  MoveL 654 to (53.54, -49.32, -190) mm, rotated rx 43.39 ry 15.84 rz 65.61 deg; joints [-1.413, -9.575, 78.286, 154.561, 95.246, 24.079, 178.286]
  MoveL 655 to (54.01, -49.44, -189.99) mm, rotated rx 43.39 ry 15.84 rz 65.61 deg; joints [-1.428, -9.587, 78.293, 154.547, 95.245, 24.086, 178.286]
  MoveL 656 to (54.51, -49.57, -189.99) mm, rotated rx 43.39 ry 15.84 rz 65.61 deg; joints [-1.445, -9.599, 78.299, 154.532, 95.243, 24.093, 178.286]
  MoveL 657 to (55.01, -49.69, -189.98) mm, rotated rx 43.39 ry 15.84 rz 65.61 deg; joints [-1.461, -9.611, 78.308, 154.518, 95.241, 24.101, 178.286]
  MoveL 658 to (55.49, -49.8, -189.95) mm, rotated rx 43.39 ry 15.84 rz 65.61 deg; joints [-1.477, -9.625, 78.317, 154.504, 95.24, 24.107, 178.286]
  MoveL 659 to (55.99, -49.92, -189.94) mm, rotated rx 43.39 ry 15.84 rz 65.61 deg; joints [-1.494, -9.637, 78.325, 154.489, 95.239, 24.115, 178.286]
  MoveL 660 to (58.53, -50.59, -189.94) mm, rotated rx 43.39 ry 15.84 rz 65.61 deg; joints [-1.578, -9.696, 78.356, 154.414, 95.227, 24.155, 178.286]
  MoveL 661 to (59.92, -51.02, -190.02) mm, rotated rx 43.39 ry 15.84 rz 65.61 deg; joints [-1.625, -9.722, 78.36, 154.372, 95.215, 24.18, 178.286]
  MoveL 662 to (61.01, -51.51, -190.27) mm, rotated rx 43.39 ry 15.84 rz 65.61 deg; joints [-1.665, -9.727, 78.336, 154.337, 95.194, 24.206, 178.286]
  MoveL 663 to (61.81, -52.06, -190.69) mm, rotated rx 43.39 ry 15.84 rz 65.61 deg; joints [-1.698, -9.714, 78.284, 154.31, 95.165, 24.233, 178.286]
  MoveL 664 to (62.32, -52.66, -191.27) mm, rotated rx 43.39 ry 15.84 rz 65.61 deg; joints [-1.723, -9.68, 78.204, 154.289, 95.127, 24.262, 178.286]
  MoveL 665 to (62.53, -53.32, -192.02) mm, rotated rx 43.39 ry 15.84 rz 65.61 deg; joints [-1.74, -9.627, 78.096, 154.275, 95.08, 24.292, 178.286]
  MoveL 666 to (62.45, -54.04, -192.93) mm, rotated rx 43.39 ry 15.84 rz 65.61 deg; joints [-1.751, -9.554, 77.959, 154.268, 95.024, 24.323, 178.286]
  MoveL 667 to (61.4, -55.64, -195.26) mm, rotated rx 43.39 ry 15.84 rz 65.61 deg; joints [-1.749, -9.349, 77.601, 154.276, 94.886, 24.389, 178.286]
  MoveL 668 to (59.59, -57.02, -197.61) mm, rotated rx 43.39 ry 15.84 rz 65.61 deg; joints [-1.722, -9.124, 77.232, 154.305, 94.752, 24.443, 178.286]
  MoveL 669 to (57.44, -57.73, -199.32) mm, rotated rx 43.39 ry 15.84 rz 65.61 deg; joints [-1.675, -8.942, 76.96, 154.351, 94.662, 24.466, 178.286]
  MoveL 670 to (56.23, -57.83, -199.93) mm, rotated rx 43.39 ry 15.84 rz 65.61 deg; joints [-1.643, -8.868, 76.859, 154.38, 94.635, 24.466, 178.286]
  MoveL 671 to (54.93, -57.77, -200.39) mm, rotated rx 43.39 ry 15.84 rz 65.61 deg; joints [-1.607, -8.803, 76.783, 154.413, 94.618, 24.459, 178.286]
  MoveL 672 to (52.09, -57.13, -200.82) mm, rotated rx 43.39 ry 15.84 rz 65.61 deg; joints [-1.518, -8.707, 76.704, 154.492, 94.619, 24.422, 178.286]
  MoveL 673 to (51.13, -56.82, -200.85) mm, rotated rx 43.39 ry 15.84 rz 65.61 deg; joints [-1.487, -8.683, 76.694, 154.52, 94.627, 24.405, 178.286]
  MoveL 674 to (48.7, -55.83, -200.85) mm, rotated rx 43.39 ry 15.84 rz 65.61 deg; joints [-1.406, -8.632, 76.694, 154.591, 94.659, 24.356, 178.286]
  MoveL 675 to (47.75, -55.49, -200.91) mm, rotated rx 43.39 ry 15.84 rz 65.61 deg; joints [-1.376, -8.608, 76.685, 154.618, 94.669, 24.339, 178.286]
  MoveL 676 to (46.78, -55.1, -200.91) mm, rotated rx 43.39 ry 15.84 rz 65.61 deg; joints [-1.343, -8.587, 76.685, 154.646, 94.682, 24.319, 178.286]
  MoveL 677 to (46.33, -54.92, -200.92) mm, rotated rx 43.39 ry 15.84 rz 65.61 deg; joints [-1.328, -8.577, 76.683, 154.66, 94.687, 24.31, 178.286]
  MoveL 678 to (45.93, -54.78, -200.94) mm, rotated rx 43.39 ry 15.84 rz 65.61 deg; joints [-1.315, -8.566, 76.679, 154.671, 94.691, 24.303, 178.286]
  MoveL 679 to (45.49, -54.62, -200.95) mm, rotated rx 43.39 ry 15.84 rz 65.61 deg; joints [-1.301, -8.556, 76.677, 154.684, 94.696, 24.295, 178.286]
  MoveL 680 to (43.06, -53.64, -200.96) mm, rotated rx 43.39 ry 15.84 rz 65.61 deg; joints [-1.22, -8.504, 76.675, 154.755, 94.728, 24.246, 178.286]
  MoveL 681 to (42.6, -53.46, -200.98) mm, rotated rx 43.39 ry 15.84 rz 65.61 deg; joints [-1.205, -8.493, 76.672, 154.768, 94.733, 24.238, 178.286]
  MoveL 682 to (42.16, -53.33, -201.02) mm, rotated rx 43.39 ry 15.84 rz 65.61 deg; joints [-1.191, -8.48, 76.664, 154.781, 94.736, 24.231, 178.286]
  MoveL 683 to (41.73, -53.23, -201.06) mm, rotated rx 43.39 ry 15.84 rz 65.61 deg; joints [-1.177, -8.467, 76.654, 154.793, 94.736, 24.225, 178.286]
  MoveL 684 to (41.3, -53.17, -201.09) mm, rotated rx 43.39 ry 15.84 rz 65.61 deg; joints [-1.163, -8.454, 76.641, 154.805, 94.734, 24.22, 178.286]
  MoveL 685 to (40.86, -53.17, -201.11) mm, rotated rx 43.39 ry 15.84 rz 65.61 deg; joints [-1.149, -8.441, 76.624, 154.818, 94.728, 24.217, 178.286]
  MoveL 686 to (40.42, -53.22, -201.11) mm, rotated rx 43.39 ry 15.84 rz 65.61 deg; joints [-1.135, -8.428, 76.603, 154.831, 94.719, 24.216, 178.286]
  MoveL 687 to (41.18, -53.27, -201.85) mm, rotated rx 43.39 ry 15.84 rz 65.61 deg; joints [-1.169, -8.398, 76.567, 154.8, 94.718, 24.23, 178.286]
  MoveL 688 to (39.84, -53.8, -202.4) mm, rotated rx 43.39 ry 15.84 rz 65.61 deg; joints [-1.134, -8.317, 76.427, 154.834, 94.66, 24.243, 178.286]
  MoveL 689 to (38.37, -54.3, -202.83) mm, rotated rx 43.39 ry 15.84 rz 65.61 deg; joints [-1.092, -8.241, 76.296, 154.874, 94.603, 24.253, 178.286]
  MoveL 690 to (36.66, -54.77, -203.13) mm, rotated rx 43.39 ry 15.84 rz 65.61 deg; joints [-1.042, -8.167, 76.166, 154.921, 94.545, 24.259, 178.286]
  MoveL 691 to (34.69, -55.23, -203.32) mm, rotated rx 43.39 ry 15.84 rz 65.61 deg; joints [-0.981, -8.093, 76.038, 154.978, 94.486, 24.261, 178.286]
  MoveL 692 to (32.65, -55.69, -203.51) mm, rotated rx 43.39 ry 15.84 rz 65.61 deg; joints [-0.918, -8.017, 75.905, 155.036, 94.424, 24.264, 178.286]
  MoveL 693 to (30.56, -56.15, -203.63) mm, rotated rx 43.39 ry 15.84 rz 65.61 deg; joints [-0.853, -7.945, 75.777, 155.097, 94.364, 24.265, 178.286]
  MoveL 694 to (28.48, -56.61, -203.86) mm, rotated rx 43.39 ry 15.84 rz 65.61 deg; joints [-0.789, -7.864, 75.639, 155.156, 94.301, 24.268, 178.286]
  MoveL 695 to (26.39, -57.06, -203.97) mm, rotated rx 43.39 ry 15.84 rz 65.61 deg; joints [-0.724, -7.792, 75.511, 155.216, 94.24, 24.268, 178.286]
  MoveL 696 to (24.31, -57.5, -204.09) mm, rotated rx 43.39 ry 15.84 rz 65.61 deg; joints [-0.659, -7.719, 75.382, 155.277, 94.179, 24.269, 178.286]
  MoveL 697 to (22.22, -57.95, -204.21) mm, rotated rx 43.39 ry 15.84 rz 65.61 deg; joints [-0.593, -7.646, 75.254, 155.337, 94.118, 24.27, 178.286]
  MoveL 698 to (20.13, -58.39, -204.44) mm, rotated rx 43.39 ry 15.84 rz 65.61 deg; joints [-0.53, -7.565, 75.115, 155.396, 94.056, 24.272, 178.286]
  MoveL 699 to (18.04, -58.83, -204.56) mm, rotated rx 43.39 ry 15.84 rz 65.61 deg; joints [-0.465, -7.491, 74.985, 155.456, 93.994, 24.273, 178.286]
  MoveL 700 to (16.05, -59.31, -204.67) mm, rotated rx 43.39 ry 15.84 rz 65.61 deg; joints [-0.403, -7.421, 74.856, 155.514, 93.931, 24.275, 178.286]
  MoveL 701 to (14.12, -59.88, -204.87) mm, rotated rx 43.39 ry 15.84 rz 65.61 deg; joints [-0.345, -7.343, 74.712, 155.568, 93.862, 24.283, 178.286]
  MoveL 702 to (11.66, -60.37, -205.01) mm, rotated rx 43.39 ry 15.84 rz 65.61 deg; joints [-0.268, -7.257, 74.561, 155.638, 93.79, 24.282, 178.286]
  MoveL 703 to (9.24, -60.72, -205.09) mm, rotated rx 43.39 ry 15.84 rz 65.61 deg; joints [-0.192, -7.176, 74.427, 155.708, 93.729, 24.278, 178.286]
  MoveL 704 to (6.99, -61.11, -205.13) mm, rotated rx 43.39 ry 15.84 rz 65.61 deg; joints [-0.121, -7.104, 74.299, 155.774, 93.668, 24.275, 178.286]
  MoveL 705 to (4.97, -61.51, -205.17) mm, rotated rx 43.39 ry 15.84 rz 65.61 deg; joints [-0.058, -7.037, 74.179, 155.832, 93.609, 24.275, 178.286]
  MoveL 706 to (3.05, -61.9, -205.29) mm, rotated rx 43.39 ry 15.84 rz 65.61 deg; joints [0.002, -6.968, 74.057, 155.887, 93.552, 24.275, 178.286]
  MoveL 707 to (1.06, -62.31, -205.35) mm, rotated rx 43.39 ry 15.84 rz 65.61 deg; joints [0.064, -6.9, 73.935, 155.944, 93.492, 24.275, 178.286]
  MoveL 708 to (-1.02, -62.73, -205.43) mm, rotated rx 43.39 ry 15.84 rz 65.61 deg; joints [0.129, -6.828, 73.806, 156.004, 93.43, 24.275, 178.286]
  MoveL 709 to (-2.97, -63.11, -205.61) mm, rotated rx 43.39 ry 15.84 rz 65.61 deg; joints [0.188, -6.753, 73.678, 156.058, 93.371, 24.276, 178.286]
  MoveL 710 to (-4.85, -63.44, -205.92) mm, rotated rx 43.39 ry 15.84 rz 65.61 deg; joints [0.243, -6.672, 73.545, 156.109, 93.315, 24.277, 178.286]
  MoveL 711 to (-5.66, -63.15, -206.96) mm, rotated rx 43.39 ry 15.84 rz 65.61 deg; joints [0.256, -6.583, 73.453, 156.121, 93.31, 24.274, 178.286]
  MoveL 712 to (-5.43, -63.04, -207.48) mm, rotated rx 43.39 ry 15.84 rz 65.61 deg; joints [0.242, -6.557, 73.43, 156.108, 93.315, 24.277, 178.286]
  MoveL 713 to (-5.42, -63.02, -207.8) mm, rotated rx 43.39 ry 15.84 rz 65.61 deg; joints [0.238, -6.536, 73.405, 156.105, 93.313, 24.28, 178.286]
  MoveL 714 to (-5.63, -63.08, -207.96) mm, rotated rx 43.39 ry 15.84 rz 65.61 deg; joints [0.242, -6.518, 73.378, 156.109, 93.304, 24.282, 178.286]
  MoveL 715 to (-6.01, -63.26, -208) mm, rotated rx 43.39 ry 15.84 rz 65.61 deg; joints [0.254, -6.501, 73.343, 156.119, 93.285, 24.286, 178.286]
  MoveL 716 to (-6.45, -63.53, -208.02) mm, rotated rx 43.39 ry 15.84 rz 65.61 deg; joints [0.267, -6.483, 73.298, 156.132, 93.259, 24.292, 178.286]
  MoveL 717 to (-6.91, -63.91, -208.03) mm, rotated rx 43.39 ry 15.84 rz 65.61 deg; joints [0.281, -6.462, 73.243, 156.145, 93.226, 24.301, 178.286]
  MoveL 718 to (-7.38, -64.34, -208.04) mm, rotated rx 43.39 ry 15.84 rz 65.61 deg; joints [0.294, -6.441, 73.185, 156.158, 93.189, 24.311, 178.286]
  MoveL 719 to (-9.94, -66.96, -208.04) mm, rotated rx 43.39 ry 15.84 rz 65.61 deg; joints [0.369, -6.321, 72.838, 156.23, 92.969, 24.376, 178.286]
  MoveL 720 to (-10.26, -67.26, -208.07) mm, rotated rx 43.39 ry 15.84 rz 65.61 deg; joints [0.378, -6.305, 72.794, 156.239, 92.943, 24.383, 178.286]
  MoveL 721 to (-10.6, -67.6, -208.08) mm, rotated rx 43.39 ry 15.84 rz 65.61 deg; joints [0.388, -6.288, 72.748, 156.248, 92.914, 24.392, 178.286]
  MoveL 722 to (-10.97, -67.97, -208.08) mm, rotated rx 43.39 ry 15.84 rz 65.61 deg; joints [0.399, -6.271, 72.697, 156.259, 92.882, 24.401, 178.286]
  MoveL 723 to (-11.32, -68.31, -208.1) mm, rotated rx 43.39 ry 15.84 rz 65.61 deg; joints [0.409, -6.253, 72.65, 156.268, 92.853, 24.409, 178.286]
  MoveL 724 to (-11.67, -68.63, -208.14) mm, rotated rx 43.39 ry 15.84 rz 65.61 deg; joints [0.419, -6.235, 72.603, 156.278, 92.826, 24.417, 178.286]
  MoveL 725 to (-12, -68.9, -208.2) mm, rotated rx 43.39 ry 15.84 rz 65.61 deg; joints [0.428, -6.217, 72.559, 156.286, 92.801, 24.424, 178.286]
  MoveL 726 to (-12.35, -69.22, -208.23) mm, rotated rx 43.39 ry 15.84 rz 65.61 deg; joints [0.437, -6.198, 72.512, 156.296, 92.773, 24.432, 178.286]
  MoveL 727 to (-12.7, -69.56, -208.25) mm, rotated rx 43.39 ry 15.84 rz 65.61 deg; joints [0.447, -6.181, 72.465, 156.305, 92.743, 24.441, 178.286]
  MoveL 728 to (-13.05, -69.92, -208.26) mm, rotated rx 43.39 ry 15.84 rz 65.61 deg; joints [0.458, -6.164, 72.416, 156.315, 92.713, 24.45, 178.286]
  MoveL 729 to (-13.42, -70.29, -208.26) mm, rotated rx 43.39 ry 15.84 rz 65.61 deg; joints [0.468, -6.147, 72.366, 156.325, 92.681, 24.459, 178.286]
  MoveL 730 to (-15.66, -72.17, -208.6) mm, rotated rx 43.39 ry 15.84 rz 65.61 deg; joints [0.53, -6.024, 72.069, 156.384, 92.511, 24.506, 178.286]
  MoveL 731 to (-16.79, -72.81, -209.04) mm, rotated rx 43.39 ry 15.84 rz 65.61 deg; joints [0.559, -5.949, 71.925, 156.411, 92.443, 24.523, 178.286]
  MoveL 732 to (-17.93, -73.25, -209.64) mm, rotated rx 43.39 ry 15.84 rz 65.61 deg; joints [0.586, -5.866, 71.784, 156.436, 92.386, 24.536, 178.286]
  MoveL 733 to (-20.24, -73.54, -211.37) mm, rotated rx 43.39 ry 15.84 rz 65.61 deg; joints [0.636, -5.675, 71.513, 156.482, 92.305, 24.549, 178.286]
  MoveL 734 to (-22.59, -73.04, -213.8) mm, rotated rx 43.39 ry 15.84 rz 65.61 deg; joints [0.68, -5.448, 71.254, 156.522, 92.268, 24.546, 178.286]
  MoveL 735 to (-24.34, -72, -216.22) mm, rotated rx 43.39 ry 15.84 rz 65.61 deg; joints [0.707, -5.249, 71.069, 156.546, 92.277, 24.53, 178.286]
  MoveL 736 to (-24.77, -71.39, -217.17) mm, rotated rx 43.39 ry 15.84 rz 65.61 deg; joints [0.71, -5.182, 71.027, 156.548, 92.299, 24.519, 178.286]
  MoveL 737 to (-24.89, -70.7, -217.95) mm, rotated rx 43.39 ry 15.84 rz 65.61 deg; joints [0.705, -5.138, 71.02, 156.544, 92.334, 24.505, 178.286]
  MoveL 738 to (-24.83, -70.34, -218.27) mm, rotated rx 43.39 ry 15.84 rz 65.61 deg; joints [0.701, -5.124, 71.029, 156.539, 92.356, 24.498, 178.286]
  MoveL 739 to (-24.7, -69.95, -218.55) mm, rotated rx 43.39 ry 15.84 rz 65.61 deg; joints [0.694, -5.115, 71.047, 156.533, 92.381, 24.49, 178.286]
  MoveL 740 to (-24.22, -69.13, -218.99) mm, rotated rx 43.39 ry 15.84 rz 65.61 deg; joints [0.675, -5.115, 71.108, 156.515, 92.44, 24.473, 178.286]
  MoveL 741 to (-23.43, -68.25, -219.25) mm, rotated rx 43.39 ry 15.84 rz 65.61 deg; joints [0.649, -5.137, 71.203, 156.49, 92.511, 24.453, 178.286]
  MoveL 742 to (-22.34, -67.3, -219.33) mm, rotated rx 43.39 ry 15.84 rz 65.61 deg; joints [0.616, -5.181, 71.332, 156.459, 92.595, 24.432, 178.286]
  MoveL 743 to (-21.92, -66.97, -219.33) mm, rotated rx 43.39 ry 15.84 rz 65.61 deg; joints [0.604, -5.199, 71.38, 156.447, 92.624, 24.424, 178.286]
  MoveL 744 to (-21.55, -66.71, -219.3) mm, rotated rx 43.39 ry 15.84 rz 65.61 deg; joints [0.593, -5.216, 71.423, 156.437, 92.65, 24.418, 178.286]
  MoveL 745 to (-21.2, -66.47, -219.26) mm, rotated rx 43.39 ry 15.84 rz 65.61 deg; joints [0.583, -5.234, 71.465, 156.428, 92.673, 24.412, 178.286]
  MoveL 746 to (-20.84, -66.24, -219.2) mm, rotated rx 43.39 ry 15.84 rz 65.61 deg; joints [0.573, -5.253, 71.506, 156.418, 92.695, 24.407, 178.286]
  MoveL 747 to (-20.47, -65.98, -219.16) mm, rotated rx 43.39 ry 15.84 rz 65.61 deg; joints [0.562, -5.271, 71.549, 156.408, 92.72, 24.401, 178.286]
  MoveL 748 to (-20.06, -65.68, -219.14) mm, rotated rx 43.39 ry 15.84 rz 65.61 deg; joints [0.55, -5.29, 71.597, 156.397, 92.748, 24.393, 178.286]
  MoveL 749 to (-19.65, -65.35, -219.14) mm, rotated rx 43.39 ry 15.84 rz 65.61 deg; joints [0.538, -5.308, 71.645, 156.386, 92.778, 24.386, 178.286]
  MoveL 750 to (-19.26, -65.04, -219.14) mm, rotated rx 43.39 ry 15.84 rz 65.61 deg; joints [0.527, -5.325, 71.691, 156.375, 92.806, 24.379, 178.286]
  MoveL 751 to (-18.88, -64.76, -219.12) mm, rotated rx 43.39 ry 15.84 rz 65.61 deg; joints [0.516, -5.343, 71.735, 156.364, 92.832, 24.372, 178.286]
  MoveL 752 to (-18.53, -64.52, -219.06) mm, rotated rx 43.39 ry 15.84 rz 65.61 deg; joints [0.506, -5.361, 71.777, 156.355, 92.855, 24.366, 178.286]
  MoveL 753 to (-18.18, -64.28, -219) mm, rotated rx 43.39 ry 15.84 rz 65.61 deg; joints [0.496, -5.38, 71.819, 156.346, 92.878, 24.36, 178.286]
  MoveL 754 to (-17.79, -64.02, -218.95) mm, rotated rx 43.39 ry 15.84 rz 65.61 deg; joints [0.485, -5.4, 71.864, 156.335, 92.903, 24.354, 178.286]
  MoveL 755 to (-17.29, -63.66, -218.91) mm, rotated rx 43.39 ry 15.84 rz 65.61 deg; joints [0.471, -5.423, 71.922, 156.322, 92.937, 24.346, 178.286]
  MoveL 756 to (-16.66, -63.2, -218.89) mm, rotated rx 43.39 ry 15.84 rz 65.61 deg; joints [0.452, -5.451, 71.994, 156.304, 92.98, 24.335, 178.286]
  MoveL 757 to (-15.43, -62.22, -218.89) mm, rotated rx 43.39 ry 15.84 rz 65.61 deg; joints [0.415, -5.504, 72.136, 156.269, 93.067, 24.312, 178.286]
  MoveL 758 to (-14.77, -61.71, -218.86) mm, rotated rx 43.39 ry 15.84 rz 65.61 deg; joints [0.396, -5.535, 72.214, 156.251, 93.114, 24.3, 178.286]
  MoveL 759 to (-14.27, -61.33, -218.85) mm, rotated rx 43.39 ry 15.84 rz 65.61 deg; joints [0.381, -5.557, 72.271, 156.237, 93.148, 24.292, 178.286]
  MoveL 760 to (-13.85, -61.07, -218.84) mm, rotated rx 43.39 ry 15.84 rz 65.61 deg; joints [0.369, -5.574, 72.313, 156.225, 93.173, 24.286, 178.286]
  MoveL 761 to (-13.48, -60.88, -218.82) mm, rotated rx 43.39 ry 15.84 rz 65.61 deg; joints [0.358, -5.589, 72.348, 156.215, 93.193, 24.282, 178.286]
  MoveL 762 to (-13.28, -60.83, -218.71) mm, rotated rx 43.39 ry 15.84 rz 65.61 deg; joints [0.353, -5.603, 72.37, 156.21, 93.201, 24.281, 178.286]
  MoveL 763 to (-13.31, -60.89, -218.49) mm, rotated rx 43.39 ry 15.84 rz 65.61 deg; joints [0.357, -5.616, 72.382, 156.213, 93.199, 24.28, 178.286]
  MoveL 764 to (-13.6, -61.07, -218.14) mm, rotated rx 43.39 ry 15.84 rz 65.61 deg; joints [0.37, -5.629, 72.382, 156.225, 93.186, 24.28, 178.286]
  MoveL 765 to (-12.95, -61.51, -217.44) mm, rotated rx 43.39 ry 15.84 rz 65.61 deg; joints [0.357, -5.688, 72.429, 156.214, 93.176, 24.29, 178.286]
  MoveL 766 to (-10.95, -61.39, -217.29) mm, rotated rx 43.39 ry 15.84 rz 65.61 deg; joints [0.295, -5.759, 72.536, 156.158, 93.22, 24.297, 178.286]
  MoveL 767 to (-9.03, -61.31, -217.01) mm, rotated rx 43.39 ry 15.84 rz 65.61 deg; joints [0.238, -5.836, 72.647, 156.105, 93.26, 24.304, 178.286]
  MoveL 768 to (-7.1, -61.21, -216.73) mm, rotated rx 43.39 ry 15.84 rz 65.61 deg; joints [0.18, -5.912, 72.76, 156.052, 93.303, 24.31, 178.286]
  MoveL 769 to (-5.17, -61.1, -216.46) mm, rotated rx 43.39 ry 15.84 rz 65.61 deg; joints [0.122, -5.988, 72.872, 155.999, 93.345, 24.316, 178.286]
  MoveL 770 to (-3.14, -60.98, -216.25) mm, rotated rx 43.39 ry 15.84 rz 65.61 deg; joints [0.06, -6.064, 72.985, 155.943, 93.388, 24.323, 178.286]
  MoveL 771 to (-1.02, -60.91, -216.1) mm, rotated rx 43.39 ry 15.84 rz 65.61 deg; joints [-0.006, -6.136, 73.089, 155.883, 93.429, 24.334, 178.286]
  MoveL 772 to (1.51, -60.95, -216) mm, rotated rx 43.39 ry 15.84 rz 65.61 deg; joints [-0.086, -6.216, 73.199, 155.81, 93.469, 24.35, 178.286]
  MoveL 773 to (3.98, -60.62, -215.92) mm, rotated rx 43.39 ry 15.84 rz 65.61 deg; joints [-0.164, -6.297, 73.335, 155.739, 93.531, 24.356, 178.286]
  MoveL 774 to (6.08, -60.35, -215.81) mm, rotated rx 43.39 ry 15.84 rz 65.61 deg; joints [-0.229, -6.369, 73.453, 155.679, 93.584, 24.36, 178.286]
  MoveL 775 to (7.96, -60.15, -215.63) mm, rotated rx 43.39 ry 15.84 rz 65.61 deg; joints [-0.287, -6.439, 73.562, 155.626, 93.628, 24.364, 178.286]
  MoveL 776 to (9.99, -59.98, -215.5) mm, rotated rx 43.39 ry 15.84 rz 65.61 deg; joints [-0.35, -6.508, 73.669, 155.568, 93.673, 24.371, 178.286]
  MoveL 777 to (12.07, -59.81, -215.37) mm, rotated rx 43.39 ry 15.84 rz 65.61 deg; joints [-0.415, -6.579, 73.778, 155.509, 93.718, 24.378, 178.286]
  MoveL 778 to (14.24, -59.63, -215.3) mm, rotated rx 43.39 ry 15.84 rz 65.61 deg; joints [-0.484, -6.648, 73.885, 155.446, 93.764, 24.386, 178.286]
  MoveL 779 to (16.36, -59.45, -215.08) mm, rotated rx 43.39 ry 15.84 rz 65.61 deg; joints [-0.549, -6.726, 74.004, 155.387, 93.811, 24.392, 178.286]
  MoveL 780 to (18.49, -59.27, -214.96) mm, rotated rx 43.39 ry 15.84 rz 65.61 deg; joints [-0.616, -6.797, 74.113, 155.326, 93.857, 24.4, 178.286]
  MoveL 781 to (20.62, -59.08, -214.74) mm, rotated rx 43.39 ry 15.84 rz 65.61 deg; joints [-0.681, -6.875, 74.231, 155.266, 93.904, 24.406, 178.286]
  MoveL 782 to (22.74, -58.9, -214.63) mm, rotated rx 43.39 ry 15.84 rz 65.61 deg; joints [-0.748, -6.945, 74.339, 155.204, 93.949, 24.413, 178.286]
  MoveL 783 to (24.87, -58.69, -214.41) mm, rotated rx 43.39 ry 15.84 rz 65.61 deg; joints [-0.813, -7.023, 74.458, 155.144, 93.997, 24.419, 178.286]
  MoveL 784 to (26.99, -58.5, -214.3) mm, rotated rx 43.39 ry 15.84 rz 65.61 deg; joints [-0.88, -7.093, 74.566, 155.083, 94.042, 24.426, 178.286]
  MoveL 785 to (29.12, -58.31, -214.2) mm, rotated rx 43.39 ry 15.84 rz 65.61 deg; joints [-0.947, -7.162, 74.673, 155.022, 94.087, 24.434, 178.286]
  MoveL 786 to (31.02, -58.08, -213.96) mm, rotated rx 43.39 ry 15.84 rz 65.61 deg; joints [-1.005, -7.234, 74.785, 154.968, 94.132, 24.437, 178.286]
  MoveL 787 to (32.83, -57.82, -213.66) mm, rotated rx 43.39 ry 15.84 rz 65.61 deg; joints [-1.06, -7.309, 74.901, 154.918, 94.179, 24.438, 178.286]
  MoveL 788 to (34.61, -57.51, -213.27) mm, rotated rx 43.39 ry 15.84 rz 65.61 deg; joints [-1.112, -7.389, 75.027, 154.87, 94.229, 24.437, 178.286]
  MoveL 789 to (33.2, -57.35, -212.35) mm, rotated rx 43.39 ry 15.84 rz 65.61 deg; joints [-1.054, -7.415, 75.064, 154.922, 94.23, 24.412, 178.286]
  MoveL 790 to (33.56, -57.33, -212.29) mm, rotated rx 43.39 ry 15.84 rz 65.61 deg; joints [-1.065, -7.429, 75.084, 154.912, 94.237, 24.413, 178.286]
  MoveL 791 to (33.93, -57.34, -212.24) mm, rotated rx 43.39 ry 15.84 rz 65.61 deg; joints [-1.076, -7.443, 75.102, 154.901, 94.242, 24.415, 178.286]
  MoveL 792 to (34.34, -57.43, -212.2) mm, rotated rx 43.39 ry 15.84 rz 65.61 deg; joints [-1.089, -7.455, 75.112, 154.89, 94.242, 24.421, 178.286]
  MoveL 793 to (34.76, -57.58, -212.18) mm, rotated rx 43.39 ry 15.84 rz 65.61 deg; joints [-1.103, -7.466, 75.117, 154.878, 94.239, 24.428, 178.286]
  MoveL 794 to (35.22, -57.8, -212.17) mm, rotated rx 43.39 ry 15.84 rz 65.61 deg; joints [-1.118, -7.476, 75.115, 154.865, 94.231, 24.438, 178.286]
  MoveL 795 to (35.67, -58.04, -212.16) mm, rotated rx 43.39 ry 15.84 rz 65.61 deg; joints [-1.133, -7.485, 75.111, 154.851, 94.221, 24.449, 178.286]
  MoveL 796 to (36.59, -58.55, -212.16) mm, rotated rx 43.39 ry 15.84 rz 65.61 deg; joints [-1.164, -7.502, 75.099, 154.825, 94.2, 24.472, 178.286]
  MoveL 797 to (37.02, -58.78, -212.15) mm, rotated rx 43.39 ry 15.84 rz 65.61 deg; joints [-1.178, -7.512, 75.096, 154.812, 94.191, 24.482, 178.286]
  MoveL 798 to (37.45, -58.98, -212.1) mm, rotated rx 43.39 ry 15.84 rz 65.61 deg; joints [-1.191, -7.524, 75.098, 154.8, 94.184, 24.491, 178.286]
  MoveL 799 to (37.93, -59.19, -212.02) mm, rotated rx 43.39 ry 15.84 rz 65.61 deg; joints [-1.206, -7.539, 75.104, 154.787, 94.178, 24.501, 178.286]
  MoveL 800 to (38.45, -59.43, -211.95) mm, rotated rx 43.39 ry 15.84 rz 65.61 deg; joints [-1.223, -7.554, 75.107, 154.773, 94.169, 24.512, 178.286]
  MoveL 801 to (38.96, -59.7, -211.92) mm, rotated rx 43.39 ry 15.84 rz 65.61 deg; joints [-1.239, -7.566, 75.105, 154.758, 94.159, 24.523, 178.286]
  MoveL 802 to (39.44, -59.95, -211.91) mm, rotated rx 43.39 ry 15.84 rz 65.61 deg; joints [-1.255, -7.576, 75.1, 154.745, 94.149, 24.535, 178.286]
  MoveL 803 to (39.91, -60.22, -211.91) mm, rotated rx 43.39 ry 15.84 rz 65.61 deg; joints [-1.271, -7.585, 75.094, 154.731, 94.138, 24.547, 178.286]
  MoveL 804 to (40.82, -60.73, -211.91) mm, rotated rx 43.39 ry 15.84 rz 65.61 deg; joints [-1.301, -7.602, 75.082, 154.705, 94.117, 24.57, 178.286]
  MoveL 805 to (41.73, -61.2, -211.88) mm, rotated rx 43.39 ry 15.84 rz 65.61 deg; joints [-1.331, -7.622, 75.076, 154.678, 94.098, 24.591, 178.286]
  MoveL 806 to (44.02, -62.48, -211.88) mm, rotated rx 43.39 ry 15.84 rz 65.61 deg; joints [-1.407, -7.664, 75.045, 154.612, 94.045, 24.649, 178.286]
  MoveL 807 to (45.24, -63.25, -211.97) mm, rotated rx 43.39 ry 15.84 rz 65.61 deg; joints [-1.45, -7.68, 75.015, 154.576, 94.01, 24.684, 178.286]
  MoveL 808 to (46.16, -63.99, -212.23) mm, rotated rx 43.39 ry 15.84 rz 65.61 deg; joints [-1.484, -7.675, 74.96, 154.546, 93.97, 24.717, 178.286]
  MoveL 809 to (46.76, -64.72, -212.67) mm, rotated rx 43.39 ry 15.84 rz 65.61 deg; joints [-1.51, -7.651, 74.881, 154.524, 93.926, 24.75, 178.286]
  MoveL 810 to (46.94, -65.07, -212.96) mm, rotated rx 43.39 ry 15.84 rz 65.61 deg; joints [-1.52, -7.631, 74.833, 154.516, 93.901, 24.766, 178.286]
  MoveL 811 to (47.05, -65.42, -213.28) mm, rotated rx 43.39 ry 15.84 rz 65.61 deg; joints [-1.528, -7.606, 74.778, 154.51, 93.876, 24.781, 178.286]
  MoveL 812 to (47.02, -66.1, -214.07) mm, rotated rx 43.39 ry 15.84 rz 65.61 deg; joints [-1.539, -7.541, 74.651, 154.502, 93.822, 24.812, 178.286]
  MoveL 813 to (46.69, -66.76, -215.04) mm, rotated rx 43.39 ry 15.84 rz 65.61 deg; joints [-1.541, -7.456, 74.5, 154.502, 93.763, 24.841, 178.286]
  MoveL 814 to (45.07, -68.01, -217.49) mm, rotated rx 43.39 ry 15.84 rz 65.61 deg; joints [-1.522, -7.225, 74.124, 154.523, 93.629, 24.897, 178.286]
  MoveL 815 to (42.79, -68.84, -219.95) mm, rotated rx 43.39 ry 15.84 rz 65.61 deg; joints [-1.482, -6.981, 73.76, 154.563, 93.513, 24.934, 178.286]
  MoveL 816 to (40.43, -68.89, -221.7) mm, rotated rx 43.39 ry 15.84 rz 65.61 deg; joints [-1.428, -6.796, 73.521, 154.612, 93.456, 24.938, 178.286]
  MoveL 817 to (39.22, -68.63, -222.32) mm, rotated rx 43.39 ry 15.84 rz 65.61 deg; joints [-1.396, -6.725, 73.448, 154.64, 93.449, 24.928, 178.286]
  MoveL 818 to (37.99, -68.17, -222.76) mm, rotated rx 43.39 ry 15.84 rz 65.61 deg; joints [-1.362, -6.669, 73.407, 154.671, 93.456, 24.909, 178.286]
  MoveL 819 to (35.47, -66.68, -223.11) mm, rotated rx 43.39 ry 15.84 rz 65.61 deg; joints [-1.283, -6.6, 73.419, 154.74, 93.516, 24.846, 178.286]
  MoveL 820 to (33.36, -65.11, -223.11) mm, rotated rx 43.39 ry 15.84 rz 65.61 deg; joints [-1.212, -6.567, 73.481, 154.801, 93.59, 24.78, 178.286]
  MoveL 821 to (32.94, -64.79, -223.09) mm, rotated rx 43.39 ry 15.84 rz 65.61 deg; joints [-1.197, -6.561, 73.495, 154.814, 93.606, 24.767, 178.286]
  MoveL 822 to (32.51, -64.46, -223.06) mm, rotated rx 43.39 ry 15.84 rz 65.61 deg; joints [-1.183, -6.557, 73.513, 154.826, 93.622, 24.752, 178.286]
  MoveL 823 to (32.11, -64.16, -223.06) mm, rotated rx 43.39 ry 15.84 rz 65.61 deg; joints [-1.169, -6.552, 73.525, 154.838, 93.637, 24.74, 178.286]
  MoveL 824 to (31.75, -63.9, -223.07) mm, rotated rx 43.39 ry 15.84 rz 65.61 deg; joints [-1.157, -6.545, 73.533, 154.848, 93.649, 24.729, 178.286]
  MoveL 825 to (31.35, -63.62, -223.1) mm, rotated rx 43.39 ry 15.84 rz 65.61 deg; joints [-1.144, -6.536, 73.541, 154.859, 93.661, 24.718, 178.286]
  MoveL 826 to (30.86, -63.32, -223.17) mm, rotated rx 43.39 ry 15.84 rz 65.61 deg; joints [-1.129, -6.523, 73.544, 154.873, 93.673, 24.705, 178.286]
  MoveL 827 to (30.36, -63.02, -223.25) mm, rotated rx 43.39 ry 15.84 rz 65.61 deg; joints [-1.113, -6.509, 73.546, 154.886, 93.685, 24.693, 178.286]
  MoveL 828 to (29.89, -62.71, -223.3) mm, rotated rx 43.39 ry 15.84 rz 65.61 deg; joints [-1.098, -6.497, 73.552, 154.9, 93.699, 24.68, 178.286]
  MoveL 829 to (29.45, -62.41, -223.32) mm, rotated rx 43.39 ry 15.84 rz 65.61 deg; joints [-1.084, -6.488, 73.561, 154.912, 93.712, 24.667, 178.286]
  MoveL 830 to (29.03, -62.1, -223.33) mm, rotated rx 43.39 ry 15.84 rz 65.61 deg; joints [-1.07, -6.481, 73.571, 154.924, 93.726, 24.655, 178.286]
  MoveL 831 to (28.61, -61.79, -223.33) mm, rotated rx 43.39 ry 15.84 rz 65.61 deg; joints [-1.055, -6.474, 73.583, 154.936, 93.741, 24.642, 178.286]
  MoveL 832 to (28.14, -61.47, -223.36) mm, rotated rx 43.39 ry 15.84 rz 65.61 deg; joints [-1.04, -6.464, 73.591, 154.949, 93.755, 24.629, 178.286]
  MoveL 833 to (27.67, -61.18, -223.41) mm, rotated rx 43.39 ry 15.84 rz 65.61 deg; joints [-1.025, -6.452, 73.595, 154.963, 93.767, 24.617, 178.286]
  MoveL 834 to (27.18, -60.91, -223.48) mm, rotated rx 43.39 ry 15.84 rz 65.61 deg; joints [-1.01, -6.438, 73.596, 154.976, 93.777, 24.605, 178.286]
  MoveL 835 to (26.72, -60.7, -223.54) mm, rotated rx 43.39 ry 15.84 rz 65.61 deg; joints [-0.995, -6.424, 73.592, 154.989, 93.783, 24.596, 178.286]
  MoveL 836 to (26.29, -60.56, -223.57) mm, rotated rx 43.39 ry 15.84 rz 65.61 deg; joints [-0.981, -6.412, 73.585, 155.001, 93.786, 24.589, 178.286]
  MoveL 837 to (25.89, -60.49, -223.58) mm, rotated rx 43.39 ry 15.84 rz 65.61 deg; joints [-0.968, -6.402, 73.575, 155.013, 93.785, 24.584, 178.286]
  MoveL 838 to (25.5, -60.46, -223.58) mm, rotated rx 43.39 ry 15.84 rz 65.61 deg; joints [-0.956, -6.391, 73.563, 155.024, 93.781, 24.58, 178.286]
  MoveL 839 to (26.76, -60.73, -224.46) mm, rotated rx 43.39 ry 15.84 rz 65.61 deg; joints [-1.008, -6.363, 73.514, 154.977, 93.771, 24.607, 178.286]
  MoveL 840 to (25.16, -60.78, -224.74) mm, rotated rx 43.39 ry 15.84 rz 65.61 deg; joints [-0.96, -6.298, 73.424, 155.021, 93.741, 24.601, 178.286]
  MoveL 841 to (23.35, -60.77, -224.93) mm, rotated rx 43.39 ry 15.84 rz 65.61 deg; joints [-0.905, -6.234, 73.338, 155.072, 93.711, 24.591, 178.286]
  MoveL 842 to (21.3, -60.72, -225.07) mm, rotated rx 43.39 ry 15.84 rz 65.61 deg; joints [-0.84, -6.168, 73.251, 155.13, 93.682, 24.577, 178.286]
  MoveL 843 to (19.06, -60.64, -225.16) mm, rotated rx 43.39 ry 15.84 rz 65.61 deg; joints [-0.769, -6.099, 73.163, 155.195, 93.652, 24.56, 178.286]
  MoveL 844 to (16.92, -60.58, -225.31) mm, rotated rx 43.39 ry 15.84 rz 65.61 deg; joints [-0.702, -6.03, 73.072, 155.256, 93.622, 24.545, 178.286]
  MoveL 845 to (14.79, -60.52, -225.52) mm, rotated rx 43.39 ry 15.84 rz 65.61 deg; joints [-0.636, -5.955, 72.974, 155.316, 93.59, 24.531, 178.286]
  MoveL 846 to (12.76, -60.46, -225.64) mm, rotated rx 43.39 ry 15.84 rz 65.61 deg; joints [-0.572, -5.89, 72.889, 155.373, 93.561, 24.517, 178.286]
  MoveL 847 to (10.91, -60.42, -225.9) mm, rotated rx 43.39 ry 15.84 rz 65.61 deg; joints [-0.516, -5.82, 72.796, 155.425, 93.531, 24.507, 178.286]
  MoveL 848 to (8.84, -60.35, -226.12) mm, rotated rx 43.39 ry 15.84 rz 65.61 deg; joints [-0.452, -5.747, 72.7, 155.482, 93.5, 24.493, 178.286]
  MoveL 849 to (6.76, -60.27, -226.26) mm, rotated rx 43.39 ry 15.84 rz 65.61 deg; joints [-0.387, -5.679, 72.612, 155.541, 93.471, 24.479, 178.286]
  MoveL 850 to (4.63, -60.18, -226.36) mm, rotated rx 43.39 ry 15.84 rz 65.61 deg; joints [-0.319, -5.612, 72.524, 155.602, 93.441, 24.463, 178.286]
  MoveL 851 to (2.51, -60.11, -226.59) mm, rotated rx 43.39 ry 15.84 rz 65.61 deg; joints [-0.254, -5.537, 72.425, 155.662, 93.409, 24.449, 178.286]
  MoveL 852 to (0.37, -60, -226.85) mm, rotated rx 43.39 ry 15.84 rz 65.61 deg; joints [-0.189, -5.459, 72.326, 155.721, 93.379, 24.435, 178.286]
  MoveL 853 to (-1.76, -59.9, -226.94) mm, rotated rx 43.39 ry 15.84 rz 65.61 deg; joints [-0.121, -5.393, 72.24, 155.782, 93.35, 24.419, 178.286]
  MoveL 854 to (-3.93, -59.8, -226.98) mm, rotated rx 43.39 ry 15.84 rz 65.61 deg; joints [-0.052, -5.329, 72.155, 155.845, 93.32, 24.402, 178.286]
  MoveL 855 to (-6.04, -59.69, -227.09) mm, rotated rx 43.39 ry 15.84 rz 65.61 deg; joints [0.014, -5.262, 72.068, 155.905, 93.291, 24.387, 178.286]
  MoveL 856 to (-8.16, -59.58, -227.29) mm, rotated rx 43.39 ry 15.84 rz 65.61 deg; joints [0.08, -5.188, 71.972, 155.964, 93.26, 24.372, 178.286]
  MoveL 857 to (-10.23, -59.46, -227.63) mm, rotated rx 43.39 ry 15.84 rz 65.61 deg; joints [0.142, -5.107, 71.868, 156.021, 93.23, 24.359, 178.286]
  MoveL 858 to (-12.38, -59.31, -227.88) mm, rotated rx 43.39 ry 15.84 rz 65.61 deg; joints [0.208, -5.029, 71.769, 156.08, 93.2, 24.343, 178.286]
  MoveL 859 to (-14.51, -59.16, -228.08) mm, rotated rx 43.39 ry 15.84 rz 65.61 deg; joints [0.274, -4.955, 71.675, 156.14, 93.171, 24.328, 178.286]
  MoveL 860 to (-16.68, -59, -228.32) mm, rotated rx 43.39 ry 15.84 rz 65.61 deg; joints [0.341, -4.877, 71.577, 156.2, 93.142, 24.312, 178.286]
  MoveL 861 to (-18.83, -58.87, -228.47) mm, rotated rx 43.39 ry 15.84 rz 65.61 deg; joints [0.408, -4.806, 71.485, 156.261, 93.112, 24.296, 178.286]
  MoveL 862 to (-20.94, -58.77, -228.49) mm, rotated rx 43.39 ry 15.84 rz 65.61 deg; joints [0.475, -4.744, 71.402, 156.322, 93.081, 24.28, 178.286]
  MoveL 863 to (-21.44, -58.38, -229.15) mm, rotated rx 43.39 ry 15.84 rz 65.61 deg; joints [0.483, -4.69, 71.359, 156.33, 93.091, 24.273, 178.286]
  MoveL 864 to (-21.12, -58.31, -229.48) mm, rotated rx 43.39 ry 15.84 rz 65.61 deg; joints [0.469, -4.678, 71.351, 156.316, 93.096, 24.276, 178.286]
  MoveL 865 to (-21.08, -58.29, -229.69) mm, rotated rx 43.39 ry 15.84 rz 65.61 deg; joints [0.465, -4.666, 71.337, 156.313, 93.096, 24.278, 178.286]
  MoveL 866 to (-21.29, -58.33, -229.79) mm, rotated rx 43.39 ry 15.84 rz 65.61 deg; joints [0.47, -4.652, 71.315, 156.318, 93.088, 24.28, 178.286]
  MoveL 867 to (-21.69, -58.47, -229.81) mm, rotated rx 43.39 ry 15.84 rz 65.61 deg; joints [0.482, -4.636, 71.283, 156.329, 93.071, 24.282, 178.286]
  MoveC 868 to (-22.59, -58.94, -229.81) mm, rotated rx 43.39 ry 15.84 rz 65.61 deg; joints [0.51, -4.601, 71.201, 156.355, 93.023, 24.291, 178.286] to (-23.46, -59.47, -229.81) mm, rotated rx 43.39 ry 15.84 rz 65.61 deg; joints [0.536, -4.566, 71.114, 156.38, 92.971, 24.302, 178.286]
  MoveL 869 to (-23.46, -59.47, -229.82) mm, rotated rx 43.39 ry 15.84 rz 65.61 deg; joints [0.536, -4.566, 71.114, 156.379, 92.971, 24.302, 178.286]
  MoveL 870 to (-23.93, -59.74, -229.84) mm, rotated rx 43.39 ry 15.84 rz 65.61 deg; joints [0.55, -4.545, 71.066, 156.393, 92.944, 24.308, 178.286]
  MoveL 871 to (-24.41, -59.99, -229.89) mm, rotated rx 43.39 ry 15.84 rz 65.61 deg; joints [0.564, -4.523, 71.017, 156.406, 92.918, 24.313, 178.286]
  MoveL 872 to (-24.93, -60.26, -229.96) mm, rotated rx 43.39 ry 15.84 rz 65.61 deg; joints [0.579, -4.498, 70.964, 156.42, 92.889, 24.319, 178.286]
  MoveL 873 to (-25.45, -60.54, -230) mm, rotated rx 43.39 ry 15.84 rz 65.61 deg; joints [0.594, -4.475, 70.912, 156.434, 92.86, 24.325, 178.286]
  MoveL 874 to (-26.49, -61.16, -230.02) mm, rotated rx 43.39 ry 15.84 rz 65.61 deg; joints [0.626, -4.431, 70.807, 156.463, 92.799, 24.338, 178.286]
  MoveL 875 to (-26.98, -61.42, -230.05) mm, rotated rx 43.39 ry 15.84 rz 65.61 deg; joints [0.64, -4.41, 70.757, 156.477, 92.771, 24.344, 178.286]
  MoveL 876 to (-27.41, -61.63, -230.13) mm, rotated rx 43.39 ry 15.84 rz 65.61 deg; joints [0.652, -4.388, 70.713, 156.488, 92.748, 24.349, 178.286]
  MoveL 877 to (-27.81, -61.81, -230.21) mm, rotated rx 43.39 ry 15.84 rz 65.61 deg; joints [0.663, -4.367, 70.671, 156.498, 92.728, 24.353, 178.286]
  MoveL 878 to (-28.19, -61.99, -230.28) mm, rotated rx 43.39 ry 15.84 rz 65.61 deg; joints [0.674, -4.348, 70.631, 156.508, 92.707, 24.357, 178.286]
  MoveL 879 to (-28.59, -62.21, -230.31) mm, rotated rx 43.39 ry 15.84 rz 65.61 deg; joints [0.685, -4.33, 70.591, 156.519, 92.685, 24.362, 178.286]
  MoveL 880 to (-30.83, -63.57, -230.31) mm, rotated rx 43.39 ry 15.84 rz 65.61 deg; joints [0.753, -4.238, 70.364, 156.582, 92.55, 24.391, 178.286]
  MoveL 881 to (-33.44, -64.84, -230.66) mm, rotated rx 43.39 ry 15.84 rz 65.61 deg; joints [0.827, -4.112, 70.098, 156.652, 92.41, 24.418, 178.286]
  MoveL 882 to (-34.67, -65.19, -231.09) mm, rotated rx 43.39 ry 15.84 rz 65.61 deg; joints [0.86, -4.038, 69.972, 156.682, 92.356, 24.427, 178.286]
  MoveL 883 to (-35.86, -65.35, -231.69) mm, rotated rx 43.39 ry 15.84 rz 65.61 deg; joints [0.889, -3.957, 69.851, 156.708, 92.314, 24.432, 178.286]
  MoveL 884 to (-37, -65.33, -232.47) mm, rotated rx 43.39 ry 15.84 rz 65.61 deg; joints [0.915, -3.869, 69.734, 156.732, 92.284, 24.434, 178.286]
  MoveL 885 to (-38.08, -65.11, -233.42) mm, rotated rx 43.39 ry 15.84 rz 65.61 deg; joints [0.938, -3.774, 69.622, 156.753, 92.264, 24.432, 178.286]
  MoveL 886 to (-40.11, -64.12, -235.83) mm, rotated rx 43.39 ry 15.84 rz 65.61 deg; joints [0.973, -3.563, 69.411, 156.785, 92.259, 24.418, 178.286]
  MoveL 887 to (-41.43, -62.75, -238.25) mm, rotated rx 43.39 ry 15.84 rz 65.61 deg; joints [0.988, -3.38, 69.267, 156.797, 92.292, 24.398, 178.286]
  MoveL 888 to (-41.65, -62.07, -239.19) mm, rotated rx 43.39 ry 15.84 rz 65.61 deg; joints [0.984, -3.32, 69.237, 156.793, 92.321, 24.387, 178.286]
  MoveL 889 to (-41.56, -61.4, -239.97) mm, rotated rx 43.39 ry 15.84 rz 65.61 deg; joints [0.973, -3.281, 69.236, 156.783, 92.357, 24.376, 178.286]
  MoveL 890 to (-41.4, -61.06, -240.29) mm, rotated rx 43.39 ry 15.84 rz 65.61 deg; joints [0.965, -3.269, 69.246, 156.775, 92.379, 24.371, 178.286]
  MoveL 891 to (-41.16, -60.73, -240.57) mm, rotated rx 43.39 ry 15.84 rz 65.61 deg; joints [0.954, -3.263, 69.263, 156.765, 92.402, 24.365, 178.286]
  MoveL 892 to (-40.47, -60.07, -241.01) mm, rotated rx 43.39 ry 15.84 rz 65.61 deg; joints [0.929, -3.266, 69.32, 156.741, 92.455, 24.354, 178.286]
  MoveL 893 to (-39.48, -59.41, -241.26) mm, rotated rx 43.39 ry 15.84 rz 65.61 deg; joints [0.896, -3.291, 69.404, 156.711, 92.515, 24.342, 178.286]
  MoveL 894 to (-38.18, -58.75, -241.35) mm, rotated rx 43.39 ry 15.84 rz 65.61 deg; joints [0.856, -3.336, 69.517, 156.673, 92.584, 24.331, 178.286]
  MoveL 895 to (-37.7, -58.53, -241.35) mm, rotated rx 43.39 ry 15.84 rz 65.61 deg; joints [0.841, -3.355, 69.559, 156.66, 92.608, 24.327, 178.286]
  MoveL 896 to (-37.28, -58.37, -241.32) mm, rotated rx 43.39 ry 15.84 rz 65.61 deg; joints [0.829, -3.373, 69.597, 156.649, 92.628, 24.324, 178.286]
  MoveL 897 to (-36.89, -58.23, -241.26) mm, rotated rx 43.39 ry 15.84 rz 65.61 deg; joints [0.817, -3.391, 69.633, 156.638, 92.646, 24.321, 178.286]
  MoveL 898 to (-36.5, -58.1, -241.19) mm, rotated rx 43.39 ry 15.84 rz 65.61 deg; joints [0.806, -3.41, 69.669, 156.628, 92.663, 24.318, 178.286]
  MoveL 899 to (-36.09, -57.95, -241.14) mm, rotated rx 43.39 ry 15.84 rz 65.61 deg; joints [0.794, -3.429, 69.706, 156.617, 92.682, 24.315, 178.286]
  MoveL 900 to (-35.62, -57.75, -241.12) mm, rotated rx 43.39 ry 15.84 rz 65.61 deg; joints [0.78, -3.448, 69.747, 156.603, 92.705, 24.312, 178.286]
  MoveL 901 to (-30.4, -55.39, -241.12) mm, rotated rx 43.39 ry 15.84 rz 65.61 deg; joints [0.621, -3.648, 70.202, 156.455, 92.964, 24.269, 178.286]
  MoveL 902 to (-29.7, -55.09, -241.1) mm, rotated rx 43.39 ry 15.84 rz 65.61 deg; joints [0.599, -3.675, 70.263, 156.435, 92.997, 24.263, 178.286]
  MoveL 903 to (-29.08, -54.86, -241.1) mm, rotated rx 43.39 ry 15.84 rz 65.61 deg; joints [0.58, -3.699, 70.313, 156.418, 93.025, 24.259, 178.286]
  MoveL 904 to (-28.52, -54.74, -241.08) mm, rotated rx 43.39 ry 15.84 rz 65.61 deg; joints [0.563, -3.718, 70.35, 156.402, 93.043, 24.259, 178.286]
  MoveL 905 to (-27.98, -54.7, -241.04) mm, rotated rx 43.39 ry 15.84 rz 65.61 deg; joints [0.546, -3.738, 70.381, 156.387, 93.056, 24.26, 178.286]
  MoveL 906 to (-27.65, -54.73, -240.88) mm, rotated rx 43.39 ry 15.84 rz 65.61 deg; joints [0.538, -3.759, 70.406, 156.379, 93.063, 24.261, 178.286]
  MoveL 907 to (-27.65, -54.76, -240.57) mm, rotated rx 43.39 ry 15.84 rz 65.61 deg; joints [0.542, -3.779, 70.431, 156.383, 93.065, 24.258, 178.286]
  MoveL 908 to (-28.02, -54.77, -240.09) mm, rotated rx 43.39 ry 15.84 rz 65.61 deg; joints [0.56, -3.802, 70.457, 156.399, 93.065, 24.251, 178.286]
  MoveL 909 to (-27.79, -55.35, -239.12) mm, rotated rx 43.39 ry 15.84 rz 65.61 deg; joints [0.564, -3.866, 70.498, 156.403, 93.044, 24.258, 178.286]
  MoveL 910 to (-25.95, -55.71, -238.82) mm, rotated rx 43.39 ry 15.84 rz 65.61 deg; joints [0.508, -3.936, 70.572, 156.352, 93.057, 24.277, 178.286]
  MoveL 911 to (-24.02, -56.06, -238.61) mm, rotated rx 43.39 ry 15.84 rz 65.61 deg; joints [0.448, -4.001, 70.642, 156.299, 93.07, 24.297, 178.286]
  MoveL 912 to (-21.93, -56.43, -238.48) mm, rotated rx 43.39 ry 15.84 rz 65.61 deg; joints [0.382, -4.066, 70.71, 156.239, 93.083, 24.32, 178.286]
  MoveL 913 to (-17.72, -57.13, -238.48) mm, rotated rx 43.39 ry 15.84 rz 65.61 deg; joints [0.246, -4.179, 70.827, 156.117, 93.109, 24.367, 178.286]
  MoveL 914 to (-15.76, -57.46, -238.39) mm, rotated rx 43.39 ry 15.84 rz 65.61 deg; joints [0.184, -4.237, 70.888, 156.061, 93.122, 24.389, 178.286]
  MoveL 915 to (-13.66, -57.81, -238.39) mm, rotated rx 43.39 ry 15.84 rz 65.61 deg; joints [0.116, -4.293, 70.946, 155.999, 93.134, 24.413, 178.286]
  MoveL 916 to (-11.54, -58.27, -238.39) mm, rotated rx 43.39 ry 15.84 rz 65.61 deg; joints [0.047, -4.348, 70.994, 155.938, 93.139, 24.44, 178.286]
  MoveL 917 to (-9.07, -58.84, -238.21) mm, rotated rx 43.39 ry 15.84 rz 65.61 deg; joints [-0.031, -4.423, 71.062, 155.868, 93.145, 24.472, 178.286]
  MoveL 918 to (-6.85, -59.08, -237.98) mm, rotated rx 43.39 ry 15.84 rz 65.61 deg; joints [-0.1, -4.5, 71.153, 155.806, 93.17, 24.491, 178.286]
  MoveL 919 to (-4.7, -59.34, -237.86) mm, rotated rx 43.39 ry 15.84 rz 65.61 deg; joints [-0.168, -4.567, 71.23, 155.745, 93.19, 24.511, 178.286]
  MoveL 920 to (-2.59, -59.69, -237.75) mm, rotated rx 43.39 ry 15.84 rz 65.61 deg; joints [-0.235, -4.63, 71.295, 155.685, 93.203, 24.534, 178.286]
  MoveL 921 to (-0.49, -60.04, -237.54) mm, rotated rx 43.39 ry 15.84 rz 65.61 deg; joints [-0.3, -4.7, 71.37, 155.626, 93.218, 24.556, 178.286]
  MoveL 922 to (1.62, -60.38, -237.43) mm, rotated rx 43.39 ry 15.84 rz 65.61 deg; joints [-0.367, -4.763, 71.435, 155.566, 93.23, 24.579, 178.286]
  MoveL 923 to (3.73, -60.73, -237.32) mm, rotated rx 43.39 ry 15.84 rz 65.61 deg; joints [-0.434, -4.825, 71.499, 155.506, 93.243, 24.603, 178.286]
  MoveL 924 to (5.83, -61.06, -237.11) mm, rotated rx 43.39 ry 15.84 rz 65.61 deg; joints [-0.499, -4.895, 71.574, 155.447, 93.258, 24.624, 178.286]
  MoveL 925 to (7.94, -61.4, -237.01) mm, rotated rx 43.39 ry 15.84 rz 65.61 deg; joints [-0.566, -4.958, 71.638, 155.387, 93.271, 24.648, 178.286]
  MoveL 926 to (10.05, -61.73, -236.9) mm, rotated rx 43.39 ry 15.84 rz 65.61 deg; joints [-0.633, -5.02, 71.702, 155.326, 93.283, 24.671, 178.286]
  MoveL 927 to (12.15, -62.05, -236.69) mm, rotated rx 43.39 ry 15.84 rz 65.61 deg; joints [-0.699, -5.089, 71.776, 155.267, 93.299, 24.693, 178.286]
  MoveL 928 to (14.26, -62.38, -236.59) mm, rotated rx 43.39 ry 15.84 rz 65.61 deg; joints [-0.766, -5.151, 71.839, 155.207, 93.311, 24.716, 178.286]
  MoveL 929 to (16.1, -62.6, -236.33) mm, rotated rx 43.39 ry 15.84 rz 65.61 deg; joints [-0.822, -5.218, 71.915, 155.157, 93.329, 24.733, 178.286]
  MoveL 930 to (17.77, -62.74, -235.97) mm, rotated rx 43.39 ry 15.84 rz 65.61 deg; joints [-0.871, -5.288, 72.001, 155.112, 93.351, 24.744, 178.286]
  MoveL 931 to (19.29, -62.79, -235.46) mm, rotated rx 43.39 ry 15.84 rz 65.61 deg; joints [-0.913, -5.365, 72.1, 155.074, 93.378, 24.75, 178.286]
  MoveL 932 to (18.24, -62.36, -234.62) mm, rotated rx 43.39 ry 15.84 rz 65.61 deg; joints [-0.868, -5.4, 72.17, 155.113, 93.402, 24.719, 178.286]
  MoveL 933 to (18.56, -62.41, -234.59) mm, rotated rx 43.39 ry 15.84 rz 65.61 deg; joints [-0.878, -5.411, 72.18, 155.104, 93.404, 24.722, 178.286]
  MoveL 934 to (18.88, -62.5, -234.55) mm, rotated rx 43.39 ry 15.84 rz 65.61 deg; joints [-0.888, -5.421, 72.189, 155.096, 93.403, 24.727, 178.286]
  MoveL 935 to (19.2, -62.67, -234.5) mm, rotated rx 43.39 ry 15.84 rz 65.61 deg; joints [-0.898, -5.431, 72.19, 155.087, 93.397, 24.734, 178.286]
  MoveL 936 to (19.54, -62.91, -234.46) mm, rotated rx 43.39 ry 15.84 rz 65.61 deg; joints [-0.909, -5.439, 72.185, 155.077, 93.387, 24.744, 178.286]
  MoveL 937 to (19.91, -63.22, -234.43) mm, rotated rx 43.39 ry 15.84 rz 65.61 deg; joints [-0.921, -5.446, 72.173, 155.067, 93.372, 24.756, 178.286]
  MoveL 938 to (23.34, -66.46, -234.43) mm, rotated rx 43.39 ry 15.84 rz 65.61 deg; joints [-1.037, -5.488, 72.01, 154.968, 93.206, 24.884, 178.286]
  MoveL 939 to (23.65, -66.72, -234.41) mm, rotated rx 43.39 ry 15.84 rz 65.61 deg; joints [-1.047, -5.494, 72, 154.959, 93.193, 24.895, 178.286]
  MoveL 940 to (24.03, -67.08, -234.41) mm, rotated rx 43.39 ry 15.84 rz 65.61 deg; joints [-1.06, -5.499, 71.982, 154.948, 93.175, 24.909, 178.286]
  MoveL 941 to (24.8, -67.76, -234.37) mm, rotated rx 43.39 ry 15.84 rz 65.61 deg; joints [-1.085, -5.511, 71.952, 154.926, 93.141, 24.936, 178.286]
  MoveL 942 to (26.7, -69.56, -234.37) mm, rotated rx 43.39 ry 15.84 rz 65.61 deg; joints [-1.15, -5.533, 71.86, 154.871, 93.048, 25.008, 178.286]
  MoveL 943 to (27.49, -70.22, -234.35) mm, rotated rx 43.39 ry 15.84 rz 65.61 deg; joints [-1.176, -5.545, 71.831, 154.849, 93.015, 25.035, 178.286]
  MoveL 944 to (28.55, -71.2, -234.42) mm, rotated rx 43.39 ry 15.84 rz 65.61 deg; joints [-1.213, -5.553, 71.776, 154.817, 92.964, 25.075, 178.286]
  MoveL 945 to (29.31, -72.1, -234.67) mm, rotated rx 43.39 ry 15.84 rz 65.61 deg; joints [-1.242, -5.542, 71.7, 154.792, 92.912, 25.113, 178.286]
  MoveL 946 to (29.77, -72.91, -235.11) mm, rotated rx 43.39 ry 15.84 rz 65.61 deg; joints [-1.263, -5.51, 71.605, 154.774, 92.858, 25.148, 178.286]
  MoveL 947 to (29.88, -73.28, -235.4) mm, rotated rx 43.39 ry 15.84 rz 65.61 deg; joints [-1.271, -5.486, 71.55, 154.768, 92.83, 25.165, 178.286]
  MoveL 948 to (29.92, -73.63, -235.74) mm, rotated rx 43.39 ry 15.84 rz 65.61 deg; joints [-1.277, -5.458, 71.489, 154.763, 92.803, 25.181, 178.286]
  MoveL 949 to (29.77, -74.27, -236.55) mm, rotated rx 43.39 ry 15.84 rz 65.61 deg; joints [-1.284, -5.386, 71.353, 154.759, 92.746, 25.21, 178.286]
  MoveL 950 to (29.31, -74.83, -237.55) mm, rotated rx 43.39 ry 15.84 rz 65.61 deg; joints [-1.283, -5.294, 71.196, 154.761, 92.687, 25.238, 178.286]
  MoveL 951 to (27.49, -75.68, -240.1) mm, rotated rx 43.39 ry 15.84 rz 65.61 deg; joints [-1.259, -5.049, 70.821, 154.785, 92.565, 25.284, 178.286]
  MoveL 952 to (25.11, -75.98, -242.67) mm, rotated rx 43.39 ry 15.84 rz 65.61 deg; joints [-1.216, -4.797, 70.474, 154.825, 92.471, 25.309, 178.286]
  MoveL 953 to (22.83, -75.49, -244.5) mm, rotated rx 43.39 ry 15.84 rz 65.61 deg; joints [-1.166, -4.613, 70.267, 154.871, 92.442, 25.3, 178.286]
  MoveL 954 to (21.72, -74.96, -245.14) mm, rotated rx 43.39 ry 15.84 rz 65.61 deg; joints [-1.138, -4.547, 70.217, 154.896, 92.451, 25.283, 178.286]
  MoveL 955 to (20.64, -74.23, -245.6) mm, rotated rx 43.39 ry 15.84 rz 65.61 deg; joints [-1.108, -4.498, 70.202, 154.922, 92.477, 25.257, 178.286]
  MoveL 956 to (18.56, -72.18, -245.96) mm, rotated rx 43.39 ry 15.84 rz 65.61 deg; joints [-1.042, -4.45, 70.279, 154.978, 92.579, 25.18, 178.286]
  MoveL 957 to (16.54, -69.77, -245.96) mm, rotated rx 43.39 ry 15.84 rz 65.61 deg; joints [-0.973, -4.437, 70.425, 155.037, 92.711, 25.087, 178.286]
  MoveL 958 to (15.87, -69.01, -245.98) mm, rotated rx 43.39 ry 15.84 rz 65.61 deg; joints [-0.95, -4.43, 70.469, 155.056, 92.753, 25.057, 178.286]
  MoveL 959 to (15.2, -68.2, -245.98) mm, rotated rx 43.39 ry 15.84 rz 65.61 deg; joints [-0.927, -4.426, 70.517, 155.076, 92.797, 25.027, 178.286]
  MoveL 960 to (14.87, -67.82, -245.98) mm, rotated rx 43.39 ry 15.84 rz 65.61 deg; joints [-0.916, -4.423, 70.539, 155.085, 92.817, 25.012, 178.286]
  MoveL 961 to (14.44, -67.32, -246.01) mm, rotated rx 43.39 ry 15.84 rz 65.61 deg; joints [-0.902, -4.417, 70.566, 155.097, 92.844, 24.993, 178.286]
  MoveL 962 to (14.03, -66.88, -246.07) mm, rotated rx 43.39 ry 15.84 rz 65.61 deg; joints [-0.889, -4.41, 70.586, 155.108, 92.867, 24.977, 178.286]
  MoveL 963 to (13.68, -66.53, -246.14) mm, rotated rx 43.39 ry 15.84 rz 65.61 deg; joints [-0.878, -4.401, 70.598, 155.118, 92.884, 24.964, 178.286]
  MoveL 964 to (13.36, -66.19, -246.19) mm, rotated rx 43.39 ry 15.84 rz 65.61 deg; joints [-0.867, -4.394, 70.612, 155.127, 92.901, 24.951, 178.286]
  MoveL 965 to (13.04, -65.85, -246.23) mm, rotated rx 43.39 ry 15.84 rz 65.61 deg; joints [-0.857, -4.389, 70.628, 155.135, 92.919, 24.938, 178.286]
  MoveL 966 to (12.03, -64.65, -246.23) mm, rotated rx 43.39 ry 15.84 rz 65.61 deg; joints [-0.823, -4.381, 70.7, 155.165, 92.985, 24.892, 178.286]
  MoveL 967 to (11.69, -64.27, -246.24) mm, rotated rx 43.39 ry 15.84 rz 65.61 deg; joints [-0.811, -4.377, 70.719, 155.174, 93.005, 24.878, 178.286]
  MoveL 968 to (11.38, -63.96, -246.27) mm, rotated rx 43.39 ry 15.84 rz 65.61 deg; joints [-0.801, -4.372, 70.733, 155.183, 93.02, 24.866, 178.286]
  MoveL 969 to (11.09, -63.72, -246.32) mm, rotated rx 43.39 ry 15.84 rz 65.61 deg; joints [-0.792, -4.364, 70.74, 155.191, 93.032, 24.857, 178.286]
  MoveL 970 to (10.82, -63.57, -246.38) mm, rotated rx 43.39 ry 15.84 rz 65.61 deg; joints [-0.784, -4.355, 70.737, 155.198, 93.036, 24.851, 178.286]
  MoveL 971 to (10.56, -63.48, -246.45) mm, rotated rx 43.39 ry 15.84 rz 65.61 deg; joints [-0.776, -4.344, 70.729, 155.205, 93.037, 24.847, 178.286]
  MoveL 972 to (11.75, -64.54, -247.26) mm, rotated rx 43.39 ry 15.84 rz 65.61 deg; joints [-0.827, -4.304, 70.608, 155.161, 92.973, 24.9, 178.286]
  MoveL 973 to (10.07, -64, -247.66) mm, rotated rx 43.39 ry 15.84 rz 65.61 deg; joints [-0.777, -4.236, 70.553, 155.206, 92.976, 24.876, 178.286]
  MoveL 974 to (8.27, -63.47, -247.92) mm, rotated rx 43.39 ry 15.84 rz 65.61 deg; joints [-0.722, -4.175, 70.506, 155.255, 92.979, 24.85, 178.286]
  MoveL 975 to (6.35, -62.92, -248.11) mm, rotated rx 43.39 ry 15.84 rz 65.61 deg; joints [-0.661, -4.116, 70.461, 155.309, 92.982, 24.822, 178.286]
  MoveL 976 to (4.29, -62.35, -248.3) mm, rotated rx 43.39 ry 15.84 rz 65.61 deg; joints [-0.597, -4.053, 70.411, 155.366, 92.983, 24.793, 178.286]
  MoveL 977 to (2.23, -61.77, -248.39) mm, rotated rx 43.39 ry 15.84 rz 65.61 deg; joints [-0.531, -3.997, 70.372, 155.425, 92.987, 24.762, 178.286]
  MoveL 978 to (0.18, -61.19, -248.49) mm, rotated rx 43.39 ry 15.84 rz 65.61 deg; joints [-0.466, -3.941, 70.332, 155.483, 92.991, 24.732, 178.286]
  MoveL 979 to (-1.87, -60.61, -248.69) mm, rotated rx 43.39 ry 15.84 rz 65.61 deg; joints [-0.401, -3.877, 70.281, 155.541, 92.993, 24.703, 178.286]
  MoveL 980 to (-3.93, -60.02, -248.79) mm, rotated rx 43.39 ry 15.84 rz 65.61 deg; joints [-0.336, -3.82, 70.241, 155.599, 92.997, 24.672, 178.286]
  MoveL 981 to (-5.98, -59.43, -248.89) mm, rotated rx 43.39 ry 15.84 rz 65.61 deg; joints [-0.27, -3.763, 70.2, 155.658, 93, 24.641, 178.286]
  MoveL 982 to (-8.03, -58.84, -249.09) mm, rotated rx 43.39 ry 15.84 rz 65.61 deg; joints [-0.206, -3.699, 70.15, 155.715, 93.002, 24.612, 178.286]
  MoveL 983 to (-12.13, -57.65, -249.29) mm, rotated rx 43.39 ry 15.84 rz 65.61 deg; joints [-0.075, -3.585, 70.067, 155.832, 93.01, 24.552, 178.286]
  MoveL 984 to (-13.85, -57.15, -249.5) mm, rotated rx 43.39 ry 15.84 rz 65.61 deg; joints [-0.021, -3.529, 70.022, 155.88, 93.011, 24.528, 178.286]
  MoveL 985 to (-15.74, -56.64, -249.57) mm, rotated rx 43.39 ry 15.84 rz 65.61 deg; joints [0.04, -3.476, 69.981, 155.934, 93.012, 24.501, 178.286]
  MoveL 986 to (-17.74, -56.15, -249.58) mm, rotated rx 43.39 ry 15.84 rz 65.61 deg; joints [0.104, -3.425, 69.938, 155.992, 93.009, 24.473, 178.286]
  MoveL 987 to (-20.3, -55.39, -249.69) mm, rotated rx 43.39 ry 15.84 rz 65.61 deg; joints [0.187, -3.354, 69.887, 156.066, 93.014, 24.435, 178.286]
  MoveL 988 to (-22.74, -54.55, -249.78) mm, rotated rx 43.39 ry 15.84 rz 65.61 deg; joints [0.265, -3.289, 69.851, 156.136, 93.027, 24.395, 178.286]
  MoveL 989 to (-24.84, -53.89, -249.88) mm, rotated rx 43.39 ry 15.84 rz 65.61 deg; joints [0.333, -3.231, 69.811, 156.196, 93.033, 24.363, 178.286]
  MoveL 990 to (-26.8, -53.29, -250.05) mm, rotated rx 43.39 ry 15.84 rz 65.61 deg; joints [0.395, -3.171, 69.765, 156.252, 93.036, 24.335, 178.286]
  MoveL 991 to (-28.62, -52.73, -250.33) mm, rotated rx 43.39 ry 15.84 rz 65.61 deg; joints [0.451, -3.107, 69.712, 156.302, 93.037, 24.31, 178.286]
  MoveL 992 to (-30.43, -52.16, -250.62) mm, rotated rx 43.39 ry 15.84 rz 65.61 deg; joints [0.506, -3.042, 69.658, 156.351, 93.039, 24.285, 178.286]
  MoveL 993 to (-32.21, -51.56, -250.91) mm, rotated rx 43.39 ry 15.84 rz 65.61 deg; joints [0.561, -2.978, 69.608, 156.4, 93.043, 24.26, 178.286]
  MoveL 994 to (-34.11, -50.97, -251.07) mm, rotated rx 43.39 ry 15.84 rz 65.61 deg; joints [0.621, -2.92, 69.564, 156.454, 93.046, 24.233, 178.286]
  MoveL 995 to (-34.43, -50.4, -251.69) mm, rotated rx 43.39 ry 15.84 rz 65.61 deg; joints [0.625, -2.877, 69.547, 156.456, 93.069, 24.221, 178.286]
  MoveL 996 to (-34.12, -50.34, -252) mm, rotated rx 43.39 ry 15.84 rz 65.61 deg; joints [0.611, -2.866, 69.539, 156.444, 93.074, 24.225, 178.286]
  MoveL 997 to (-34.1, -50.3, -252.19) mm, rotated rx 43.39 ry 15.84 rz 65.61 deg; joints [0.608, -2.854, 69.527, 156.441, 93.074, 24.226, 178.286]
  MoveL 998 to (-34.35, -50.28, -252.29) mm, rotated rx 43.39 ry 15.84 rz 65.61 deg; joints [0.614, -2.84, 69.508, 156.447, 93.069, 24.225, 178.286]
  MoveL 999 to (-34.79, -50.33, -252.31) mm, rotated rx 43.39 ry 15.84 rz 65.61 deg; joints [0.628, -2.824, 69.482, 156.46, 93.057, 24.225, 178.286]
  MoveL 1000 to (-35.27, -50.43, -252.31) mm, rotated rx 43.39 ry 15.84 rz 65.61 deg; joints [0.643, -2.808, 69.451, 156.474, 93.042, 24.225, 178.286]
  MoveL 1001 to (-36.21, -50.72, -252.35) mm, rotated rx 43.39 ry 15.84 rz 65.61 deg; joints [0.672, -2.772, 69.379, 156.5, 93.004, 24.229, 178.286]
  MoveL 1002 to (-37.7, -51.19, -252.35) mm, rotated rx 43.39 ry 15.84 rz 65.61 deg; joints [0.718, -2.718, 69.266, 156.543, 92.943, 24.235, 178.286]
  MoveL 1003 to (-38.65, -51.45, -252.36) mm, rotated rx 43.39 ry 15.84 rz 65.61 deg; joints [0.747, -2.684, 69.197, 156.57, 92.906, 24.239, 178.286]
  MoveL 1004 to (-39.65, -51.77, -252.36) mm, rotated rx 43.39 ry 15.84 rz 65.61 deg; joints [0.778, -2.647, 69.122, 156.598, 92.866, 24.243, 178.286]
  MoveL 1005 to (-40.14, -51.92, -252.38) mm, rotated rx 43.39 ry 15.84 rz 65.61 deg; joints [0.793, -2.629, 69.084, 156.612, 92.846, 24.245, 178.286]
  MoveL 1006 to (-40.59, -52.05, -252.41) mm, rotated rx 43.39 ry 15.84 rz 65.61 deg; joints [0.807, -2.61, 69.048, 156.625, 92.827, 24.247, 178.286]
  MoveL 1007 to (-41.02, -52.16, -252.45) mm, rotated rx 43.39 ry 15.84 rz 65.61 deg; joints [0.819, -2.592, 69.014, 156.636, 92.811, 24.248, 178.286]
  MoveL 1008 to (-41.41, -52.25, -252.51) mm, rotated rx 43.39 ry 15.84 rz 65.61 deg; joints [0.831, -2.574, 68.982, 156.647, 92.796, 24.25, 178.286]
  MoveL 1009 to (-41.82, -52.35, -252.57) mm, rotated rx 43.39 ry 15.84 rz 65.61 deg; joints [0.843, -2.556, 68.948, 156.658, 92.78, 24.252, 178.286]
  MoveL 1010 to (-42.26, -52.48, -252.6) mm, rotated rx 43.39 ry 15.84 rz 65.61 deg; joints [0.856, -2.538, 68.914, 156.67, 92.763, 24.253, 178.286]
  MoveL 1011 to (-42.72, -52.61, -252.63) mm, rotated rx 43.39 ry 15.84 rz 65.61 deg; joints [0.87, -2.52, 68.878, 156.683, 92.744, 24.255, 178.286]
  MoveL 1012 to (-43.15, -52.71, -252.67) mm, rotated rx 43.39 ry 15.84 rz 65.61 deg; joints [0.882, -2.502, 68.845, 156.695, 92.728, 24.257, 178.286]
  MoveL 1013 to (-43.54, -52.79, -252.73) mm, rotated rx 43.39 ry 15.84 rz 65.61 deg; joints [0.894, -2.484, 68.813, 156.705, 92.714, 24.258, 178.286]
  MoveL 1014 to (-43.94, -52.88, -252.78) mm, rotated rx 43.39 ry 15.84 rz 65.61 deg; joints [0.906, -2.467, 68.782, 156.716, 92.699, 24.259, 178.286]
  MoveL 1015 to (-44.37, -53, -252.81) mm, rotated rx 43.39 ry 15.84 rz 65.61 deg; joints [0.919, -2.449, 68.748, 156.728, 92.682, 24.261, 178.286]
  MoveL 1016 to (-44.87, -53.15, -252.81) mm, rotated rx 43.39 ry 15.84 rz 65.61 deg; joints [0.934, -2.431, 68.71, 156.742, 92.662, 24.263, 178.286]
  MoveL 1017 to (-47.71, -53.79, -253.17) mm, rotated rx 43.39 ry 15.84 rz 65.61 deg; joints [1.018, -2.306, 68.486, 156.819, 92.556, 24.271, 178.286]
  MoveL 1018 to (-49, -53.87, -253.61) mm, rotated rx 43.39 ry 15.84 rz 65.61 deg; joints [1.052, -2.234, 68.378, 156.851, 92.518, 24.272, 178.286]
  MoveL 1019 to (-50.2, -53.78, -254.24) mm, rotated rx 43.39 ry 15.84 rz 65.61 deg; joints [1.082, -2.154, 68.273, 156.878, 92.49, 24.271, 178.286]
  MoveL 1020 to (-52.32, -53.12, -256.02) mm, rotated rx 43.39 ry 15.84 rz 65.61 deg; joints [1.128, -1.975, 68.073, 156.92, 92.464, 24.262, 178.286]
  MoveL 1021 to (-54.07, -51.82, -258.51) mm, rotated rx 43.39 ry 15.84 rz 65.61 deg; joints [1.155, -1.768, 67.885, 156.944, 92.477, 24.245, 178.286]
  MoveL 1022 to (-55.06, -50.31, -261) mm, rotated rx 43.39 ry 15.84 rz 65.61 deg; joints [1.158, -1.588, 67.751, 156.946, 92.519, 24.226, 178.286]
  MoveL 1023 to (-55.12, -49.66, -261.98) mm, rotated rx 43.39 ry 15.84 rz 65.61 deg; joints [1.149, -1.529, 67.72, 156.937, 92.546, 24.218, 178.286]
  MoveL 1024 to (-54.88, -49.07, -262.78) mm, rotated rx 43.39 ry 15.84 rz 65.61 deg; joints [1.133, -1.491, 67.713, 156.922, 92.578, 24.211, 178.286]
  MoveL 1025 to (-54.65, -48.8, -263.12) mm, rotated rx 43.39 ry 15.84 rz 65.61 deg; joints [1.122, -1.479, 67.719, 156.912, 92.596, 24.209, 178.286]
  MoveL 1026 to (-54.35, -48.54, -263.41) mm, rotated rx 43.39 ry 15.84 rz 65.61 deg; joints [1.11, -1.473, 67.731, 156.9, 92.614, 24.206, 178.286]
  MoveL 1027 to (-53.52, -48.08, -263.85) mm, rotated rx 43.39 ry 15.84 rz 65.61 deg; joints [1.079, -1.475, 67.773, 156.872, 92.656, 24.202, 178.286]
  MoveL 1028 to (-52.41, -47.68, -264.12) mm, rotated rx 43.39 ry 15.84 rz 65.61 deg; joints [1.041, -1.498, 67.839, 156.837, 92.701, 24.199, 178.286]
  MoveL 1029 to (-51, -47.34, -264.21) mm, rotated rx 43.39 ry 15.84 rz 65.61 deg; joints [0.996, -1.542, 67.93, 156.796, 92.751, 24.197, 178.286]
  MoveL 1030 to (-48.43, -46.84, -264.21) mm, rotated rx 43.39 ry 15.84 rz 65.61 deg; joints [0.916, -1.631, 68.099, 156.722, 92.837, 24.195, 178.286]
  MoveL 1031 to (-47.99, -46.77, -264.18) mm, rotated rx 43.39 ry 15.84 rz 65.61 deg; joints [0.903, -1.648, 68.129, 156.71, 92.851, 24.195, 178.286]
  MoveL 1032 to (-47.59, -46.71, -264.13) mm, rotated rx 43.39 ry 15.84 rz 65.61 deg; joints [0.891, -1.665, 68.157, 156.699, 92.864, 24.194, 178.286]
  MoveL 1033 to (-47.21, -46.67, -264.06) mm, rotated rx 43.39 ry 15.84 rz 65.61 deg; joints [0.88, -1.682, 68.185, 156.689, 92.875, 24.194, 178.286]
  MoveL 1034 to (-46.78, -46.62, -264.01) mm, rotated rx 43.39 ry 15.84 rz 65.61 deg; joints [0.867, -1.7, 68.215, 156.677, 92.889, 24.194, 178.286]
  MoveL 1035 to (-46.29, -46.54, -263.97) mm, rotated rx 43.39 ry 15.84 rz 65.61 deg; joints [0.852, -1.719, 68.249, 156.664, 92.904, 24.194, 178.286]
  MoveL 1036 to (-45.77, -46.47, -263.92) mm, rotated rx 43.39 ry 15.84 rz 65.61 deg; joints [0.836, -1.741, 68.285, 156.649, 92.92, 24.194, 178.286]
  MoveL 1037 to (-45.23, -46.37, -263.9) mm, rotated rx 43.39 ry 15.84 rz 65.61 deg; joints [0.82, -1.76, 68.32, 156.634, 92.938, 24.193, 178.286]
  MoveL 1038 to (-44.6, -46.25, -263.91) mm, rotated rx 43.39 ry 15.84 rz 65.61 deg; joints [0.8, -1.781, 68.36, 156.616, 92.959, 24.193, 178.286]
  MoveL 1039 to (-43.75, -46.05, -263.98) mm, rotated rx 43.39 ry 15.84 rz 65.61 deg; joints [0.773, -1.805, 68.412, 156.591, 92.987, 24.192, 178.286]
  MoveL 1040 to (-43.24, -45.95, -263.98) mm, rotated rx 43.39 ry 15.84 rz 65.61 deg; joints [0.757, -1.823, 68.445, 156.576, 93.004, 24.192, 178.286]
  MoveL 1041 to (-42.75, -45.86, -263.97) mm, rotated rx 43.39 ry 15.84 rz 65.61 deg; joints [0.742, -1.84, 68.477, 156.562, 93.02, 24.192, 178.286]
  MoveL 1042 to (-42.29, -45.78, -263.95) mm, rotated rx 43.39 ry 15.84 rz 65.61 deg; joints [0.727, -1.857, 68.508, 156.549, 93.035, 24.191, 178.286]
  MoveL 1043 to (-41.88, -45.73, -263.9) mm, rotated rx 43.39 ry 15.84 rz 65.61 deg; joints [0.715, -1.875, 68.537, 156.538, 93.048, 24.191, 178.286]
  MoveL 1044 to (-41.48, -45.7, -263.84) mm, rotated rx 43.39 ry 15.84 rz 65.61 deg; joints [0.703, -1.891, 68.563, 156.527, 93.059, 24.191, 178.286]
  MoveL 1045 to (-41.06, -45.7, -263.79) mm, rotated rx 43.39 ry 15.84 rz 65.61 deg; joints [0.69, -1.908, 68.587, 156.515, 93.067, 24.193, 178.286]
  MoveL 1046 to (-40.65, -45.76, -263.73) mm, rotated rx 43.39 ry 15.84 rz 65.61 deg; joints [0.678, -1.923, 68.606, 156.504, 93.072, 24.196, 178.286]
  MoveL 1047 to (-40.44, -45.85, -263.57) mm, rotated rx 43.39 ry 15.84 rz 65.61 deg; joints [0.673, -1.94, 68.622, 156.5, 93.073, 24.198, 178.286]
  MoveL 1048 to (-40.54, -45.9, -263.26) mm, rotated rx 43.39 ry 15.84 rz 65.61 deg; joints [0.68, -1.958, 68.641, 156.506, 93.072, 24.195, 178.286]
  MoveL 1049 to (-40.98, -45.92, -262.77) mm, rotated rx 43.39 ry 15.84 rz 65.61 deg; joints [0.701, -1.979, 68.664, 156.524, 93.071, 24.187, 178.286]
  MoveL 1050 to (-40.15, -46.23, -261.92) mm, rotated rx 43.39 ry 15.84 rz 65.61 deg; joints [0.684, -2.059, 68.751, 156.51, 93.08, 24.19, 178.286]
  MoveL 1051 to (-36.21, -47.88, -261.92) mm, rotated rx 43.39 ry 15.84 rz 65.61 deg; joints [0.554, -2.15, 68.777, 156.394, 93.041, 24.264, 178.286]
  MoveL 1052 to (-34.37, -48.66, -261.85) mm, rotated rx 43.39 ry 15.84 rz 65.61 deg; joints [0.494, -2.197, 68.793, 156.341, 93.023, 24.298, 178.286]
  MoveL 1053 to (-32.54, -49.45, -261.7) mm, rotated rx 43.39 ry 15.84 rz 65.61 deg; joints [0.436, -2.249, 68.816, 156.289, 93.005, 24.331, 178.286]
  MoveL 1054 to (-30.43, -50.35, -261.5) mm, rotated rx 43.39 ry 15.84 rz 65.61 deg; joints [0.369, -2.31, 68.844, 156.23, 92.985, 24.369, 178.286]
  MoveL 1055 to (-28.43, -51.21, -261.29) mm, rotated rx 43.39 ry 15.84 rz 65.61 deg; joints [0.306, -2.371, 68.873, 156.173, 92.966, 24.405, 178.286]
  MoveL 1056 to (-26.42, -52.06, -261.19) mm, rotated rx 43.39 ry 15.84 rz 65.61 deg; joints [0.241, -2.423, 68.892, 156.116, 92.946, 24.442, 178.286]
  MoveL 1057 to (-24.46, -52.89, -261.19) mm, rotated rx 43.39 ry 15.84 rz 65.61 deg; joints [0.176, -2.468, 68.903, 156.058, 92.926, 24.479, 178.286]
  MoveL 1058 to (-22.63, -53.65, -261.13) mm, rotated rx 43.39 ry 15.84 rz 65.61 deg; joints [0.117, -2.514, 68.918, 156.006, 92.907, 24.514, 178.286]
  MoveL 1059 to (-20.9, -54.38, -261.01) mm, rotated rx 43.39 ry 15.84 rz 65.61 deg; joints [0.061, -2.561, 68.937, 155.956, 92.891, 24.545, 178.286]
  MoveL 1060 to (-19.01, -55.16, -260.94) mm, rotated rx 43.39 ry 15.84 rz 65.61 deg; joints [0, -2.608, 68.953, 155.902, 92.872, 24.581, 178.286]
  MoveL 1061 to (-17.04, -55.99, -260.76) mm, rotated rx 43.39 ry 15.84 rz 65.61 deg; joints [-0.062, -2.665, 68.978, 155.847, 92.854, 24.616, 178.286]
  MoveL 1062 to (-13.1, -57.63, -260.58) mm, rotated rx 43.39 ry 15.84 rz 65.61 deg; joints [-0.189, -2.766, 69.012, 155.734, 92.814, 24.69, 178.286]
  MoveL 1063 to (-11.13, -58.44, -260.4) mm, rotated rx 43.39 ry 15.84 rz 65.61 deg; joints [-0.252, -2.822, 69.038, 155.679, 92.796, 24.726, 178.286]
  MoveL 1064 to (-9.15, -59.25, -260.22) mm, rotated rx 43.39 ry 15.84 rz 65.61 deg; joints [-0.314, -2.879, 69.063, 155.623, 92.778, 24.762, 178.286]
  MoveL 1065 to (-7.19, -60.08, -260.22) mm, rotated rx 43.39 ry 15.84 rz 65.61 deg; joints [-0.379, -2.922, 69.07, 155.566, 92.756, 24.801, 178.286]
  MoveL 1066 to (-5.21, -60.88, -260.04) mm, rotated rx 43.39 ry 15.84 rz 65.61 deg; joints [-0.442, -2.979, 69.096, 155.511, 92.738, 24.837, 178.286]
  MoveL 1067 to (-3.23, -61.68, -259.87) mm, rotated rx 43.39 ry 15.84 rz 65.61 deg; joints [-0.504, -3.035, 69.121, 155.455, 92.72, 24.873, 178.286]
  MoveL 1068 to (-1.26, -62.51, -259.87) mm, rotated rx 43.39 ry 15.84 rz 65.61 deg; joints [-0.569, -3.078, 69.127, 155.398, 92.697, 24.912, 178.286]
  MoveL 1069 to (0.56, -63.19, -259.67) mm, rotated rx 43.39 ry 15.84 rz 65.61 deg; joints [-0.626, -3.133, 69.157, 155.347, 92.685, 24.943, 178.286]
  MoveL 1070 to (2.19, -63.73, -259.35) mm, rotated rx 43.39 ry 15.84 rz 65.61 deg; joints [-0.674, -3.193, 69.204, 155.304, 92.681, 24.967, 178.286]
  MoveL 1071 to (3.66, -64.14, -258.88) mm, rotated rx 43.39 ry 15.84 rz 65.61 deg; joints [-0.716, -3.262, 69.27, 155.266, 92.686, 24.983, 178.286]
  MoveL 1072 to (2.87, -63.62, -258.12) mm, rotated rx 43.39 ry 15.84 rz 65.61 deg; joints [-0.68, -3.302, 69.355, 155.298, 92.72, 24.951, 178.286]
  MoveL 1073 to (3.23, -63.82, -258.11) mm, rotated rx 43.39 ry 15.84 rz 65.61 deg; joints [-0.692, -3.309, 69.352, 155.287, 92.712, 24.96, 178.286]
  MoveC 1074 to (5.42, -66.62, -258.11) mm, rotated rx 43.39 ry 15.84 rz 65.61 deg; joints [-0.768, -3.322, 69.179, 155.223, 92.557, 25.066, 178.286] to (7.37, -69.59, -258.11) mm, rotated rx 43.39 ry 15.84 rz 65.61 deg; joints [-0.836, -3.323, 68.977, 155.166, 92.384, 25.176, 178.286]
  MoveL 1075 to (7.37, -69.59, -258.11) mm, rotated rx 43.39 ry 15.84 rz 65.61 deg; joints [-0.836, -3.323, 68.977, 155.166, 92.384, 25.176, 178.286]
  MoveL 1076 to (7.64, -69.98, -258.09) mm, rotated rx 43.39 ry 15.84 rz 65.61 deg; joints [-0.845, -3.325, 68.953, 155.158, 92.363, 25.191, 178.286]
  MoveL 1077 to (7.9, -70.31, -258.04) mm, rotated rx 43.39 ry 15.84 rz 65.61 deg; joints [-0.853, -3.33, 68.937, 155.152, 92.345, 25.203, 178.286]
  MoveL 1078 to (8.15, -70.63, -257.98) mm, rotated rx 43.39 ry 15.84 rz 65.61 deg; joints [-0.861, -3.335, 68.922, 155.145, 92.328, 25.214, 178.286]
  MoveL 1079 to (8.41, -70.98, -257.93) mm, rotated rx 43.39 ry 15.84 rz 65.61 deg; joints [-0.869, -3.339, 68.903, 155.138, 92.309, 25.227, 178.286]
  MoveL 1080 to (8.68, -71.37, -257.9) mm, rotated rx 43.39 ry 15.84 rz 65.61 deg; joints [-0.878, -3.342, 68.881, 155.13, 92.287, 25.241, 178.286]
  MoveL 1081 to (8.98, -71.8, -257.89) mm, rotated rx 43.39 ry 15.84 rz 65.61 deg; joints [-0.888, -3.343, 68.853, 155.122, 92.263, 25.257, 178.286]
  MoveL 1082 to (9.55, -72.67, -257.89) mm, rotated rx 43.39 ry 15.84 rz 65.61 deg; joints [-0.908, -3.343, 68.793, 155.105, 92.212, 25.29, 178.286]
  MoveL 1083 to (10.31, -73.92, -257.98) mm, rotated rx 43.39 ry 15.84 rz 65.61 deg; joints [-0.936, -3.335, 68.697, 155.082, 92.137, 25.337, 178.286]
  MoveL 1084 to (10.82, -75.01, -258.26) mm, rotated rx 43.39 ry 15.84 rz 65.61 deg; joints [-0.957, -3.309, 68.588, 155.063, 92.065, 25.38, 178.286]
  MoveL 1085 to (11.09, -75.93, -258.71) mm, rotated rx 43.39 ry 15.84 rz 65.61 deg; joints [-0.973, -3.266, 68.468, 155.05, 91.998, 25.419, 178.286]
  MoveL 1086 to (11.12, -76.7, -259.35) mm, rotated rx 43.39 ry 15.84 rz 65.61 deg; joints [-0.984, -3.207, 68.336, 155.042, 91.935, 25.453, 178.286]
  MoveL 1087 to (10.9, -77.32, -260.18) mm, rotated rx 43.39 ry 15.84 rz 65.61 deg; joints [-0.989, -3.13, 68.193, 155.038, 91.875, 25.484, 178.286]
  MoveL 1088 to (10.45, -77.77, -261.18) mm, rotated rx 43.39 ry 15.84 rz 65.61 deg; joints [-0.988, -3.036, 68.037, 155.04, 91.819, 25.509, 178.286]
  MoveL 1089 to (8.81, -78.2, -263.74) mm, rotated rx 43.39 ry 15.84 rz 65.61 deg; joints [-0.969, -2.797, 67.69, 155.058, 91.717, 25.548, 178.286]
  MoveL 1090 to (6.78, -77.94, -266.3) mm, rotated rx 43.39 ry 15.84 rz 65.61 deg; joints [-0.937, -2.559, 67.39, 155.088, 91.656, 25.561, 178.286]
  MoveL 1091 to (5.82, -77.54, -267.31) mm, rotated rx 43.39 ry 15.84 rz 65.61 deg; joints [-0.918, -2.467, 67.295, 155.104, 91.65, 25.555, 178.286]
  MoveL 1092 to (4.91, -76.96, -268.13) mm, rotated rx 43.39 ry 15.84 rz 65.61 deg; joints [-0.899, -2.393, 67.237, 155.122, 91.66, 25.541, 178.286]
  MoveL 1093 to (4.04, -76.19, -268.77) mm, rotated rx 43.39 ry 15.84 rz 65.61 deg; joints [-0.878, -2.337, 67.215, 155.14, 91.687, 25.519, 178.286]
  MoveL 1094 to (3.21, -75.23, -269.23) mm, rotated rx 43.39 ry 15.84 rz 65.61 deg; joints [-0.856, -2.299, 67.23, 155.159, 91.731, 25.488, 178.286]
  MoveL 1095 to (1.67, -72.78, -269.59) mm, rotated rx 43.39 ry 15.84 rz 65.61 deg; joints [-0.807, -2.277, 67.37, 155.201, 91.87, 25.401, 178.286]
  MoveL 1096 to (1.19, -71.84, -269.59) mm, rotated rx 43.39 ry 15.84 rz 65.61 deg; joints [-0.79, -2.281, 67.44, 155.215, 91.927, 25.367, 178.286]
  MoveL 1097 to (0.95, -71.38, -269.6) mm, rotated rx 43.39 ry 15.84 rz 65.61 deg; joints [-0.781, -2.283, 67.474, 155.222, 91.955, 25.35, 178.286]
  MoveL 1098 to (0.72, -70.96, -269.62) mm, rotated rx 43.39 ry 15.84 rz 65.61 deg; joints [-0.774, -2.283, 67.503, 155.229, 91.979, 25.335, 178.286]
  MoveL 1099 to (0.5, -70.6, -269.67) mm, rotated rx 43.39 ry 15.84 rz 65.61 deg; joints [-0.767, -2.28, 67.524, 155.235, 92, 25.323, 178.286]
  MoveL 1100 to (0.29, -70.26, -269.73) mm, rotated rx 43.39 ry 15.84 rz 65.61 deg; joints [-0.76, -2.276, 67.543, 155.24, 92.019, 25.311, 178.286]
  MoveL 1101 to (0.08, -69.9, -269.77) mm, rotated rx 43.39 ry 15.84 rz 65.61 deg; joints [-0.753, -2.274, 67.564, 155.246, 92.04, 25.298, 178.286]
  MoveL 1102 to (-0.15, -69.48, -269.79) mm, rotated rx 43.39 ry 15.84 rz 65.61 deg; joints [-0.745, -2.274, 67.593, 155.252, 92.064, 25.283, 178.286]
  MoveL 1103 to (-0.38, -69.04, -269.8) mm, rotated rx 43.39 ry 15.84 rz 65.61 deg; joints [-0.737, -2.275, 67.625, 155.259, 92.091, 25.267, 178.286]
  MoveL 1104 to (-0.63, -68.55, -269.79) mm, rotated rx 43.39 ry 15.84 rz 65.61 deg; joints [-0.728, -2.278, 67.663, 155.267, 92.121, 25.249, 178.286]
  MoveL 1105 to (-0.88, -68.08, -269.8) mm, rotated rx 43.39 ry 15.84 rz 65.61 deg; joints [-0.719, -2.279, 67.697, 155.274, 92.149, 25.232, 178.286]
  MoveL 1106 to (-1.11, -67.65, -269.83) mm, rotated rx 43.39 ry 15.84 rz 65.61 deg; joints [-0.711, -2.279, 67.726, 155.281, 92.175, 25.217, 178.286]
  MoveL 1107 to (-1.35, -67.23, -269.87) mm, rotated rx 43.39 ry 15.84 rz 65.61 deg; joints [-0.704, -2.277, 67.752, 155.287, 92.199, 25.202, 178.286]
  MoveL 1108 to (-1.61, -66.8, -269.95) mm, rotated rx 43.39 ry 15.84 rz 65.61 deg; joints [-0.695, -2.272, 67.775, 155.294, 92.223, 25.187, 178.286]
  MoveL 1109 to (-1.92, -66.28, -270.01) mm, rotated rx 43.39 ry 15.84 rz 65.61 deg; joints [-0.685, -2.268, 67.806, 155.303, 92.252, 25.169, 178.286]
  MoveL 1110 to (-2.19, -65.78, -270.03) mm, rotated rx 43.39 ry 15.84 rz 65.61 deg; joints [-0.676, -2.269, 67.841, 155.311, 92.282, 25.151, 178.286]
  MoveL 1111 to (-2.44, -65.31, -270.03) mm, rotated rx 43.39 ry 15.84 rz 65.61 deg; joints [-0.667, -2.27, 67.875, 155.318, 92.31, 25.134, 178.286]
  MoveL 1112 to (-2.67, -64.85, -270.03) mm, rotated rx 43.39 ry 15.84 rz 65.61 deg; joints [-0.659, -2.272, 67.91, 155.325, 92.339, 25.117, 178.286]
  MoveL 1113 to (-2.99, -64.27, -270.04) mm, rotated rx 43.39 ry 15.84 rz 65.61 deg; joints [-0.647, -2.273, 67.95, 155.334, 92.373, 25.096, 178.286]
  MoveL 1114 to (-3.29, -63.77, -270.05) mm, rotated rx 43.39 ry 15.84 rz 65.61 deg; joints [-0.637, -2.273, 67.985, 155.343, 92.402, 25.078, 178.286]
  MoveL 1115 to (-3.57, -63.35, -270.06) mm, rotated rx 43.39 ry 15.84 rz 65.61 deg; joints [-0.627, -2.272, 68.012, 155.351, 92.426, 25.063, 178.286]
  MoveL 1116 to (-3.81, -63.1, -270.06) mm, rotated rx 43.39 ry 15.84 rz 65.61 deg; joints [-0.619, -2.27, 68.026, 155.358, 92.44, 25.053, 178.286]
  MoveL 1117 to (-4.02, -62.93, -270.06) mm, rotated rx 43.39 ry 15.84 rz 65.61 deg; joints [-0.612, -2.267, 68.033, 155.364, 92.447, 25.046, 178.286]
  MoveL 1118 to (-3.27, -63.5, -270.65) mm, rotated rx 43.39 ry 15.84 rz 65.61 deg; joints [-0.645, -2.236, 67.956, 155.336, 92.411, 25.078, 178.286]
  MoveL 1119 to (-4.55, -63.1, -271.18) mm, rotated rx 43.39 ry 15.84 rz 65.61 deg; joints [-0.61, -2.168, 67.889, 155.367, 92.407, 25.064, 178.286]
  MoveL 1120 to (-5.99, -62.51, -271.56) mm, rotated rx 43.39 ry 15.84 rz 65.61 deg; joints [-0.568, -2.109, 67.848, 155.404, 92.415, 25.041, 178.286]
  MoveL 1121 to (-7.66, -61.71, -271.82) mm, rotated rx 43.39 ry 15.84 rz 65.61 deg; joints [-0.517, -2.056, 67.828, 155.45, 92.437, 25.008, 178.286]
  MoveL 1122 to (-9.47, -60.74, -271.95) mm, rotated rx 43.39 ry 15.84 rz 65.61 deg; joints [-0.459, -2.011, 67.83, 155.501, 92.469, 24.967, 178.286]
  MoveL 1123 to (-11.32, -59.73, -272.04) mm, rotated rx 43.39 ry 15.84 rz 65.61 deg; joints [-0.399, -1.968, 67.836, 155.554, 92.504, 24.924, 178.286]
  MoveL 1124 to (-15.06, -57.68, -272.22) mm, rotated rx 43.39 ry 15.84 rz 65.61 deg; joints [-0.277, -1.882, 67.85, 155.661, 92.575, 24.838, 178.286]
  MoveL 1125 to (-16.93, -56.67, -272.4) mm, rotated rx 43.39 ry 15.84 rz 65.61 deg; joints [-0.218, -1.831, 67.847, 155.713, 92.608, 24.796, 178.286]
  MoveL 1126 to (-20.67, -54.61, -272.58) mm, rotated rx 43.39 ry 15.84 rz 65.61 deg; joints [-0.096, -1.744, 67.859, 155.82, 92.679, 24.71, 178.286]
  MoveL 1127 to (-22.54, -53.58, -272.76) mm, rotated rx 43.39 ry 15.84 rz 65.61 deg; joints [-0.037, -1.693, 67.856, 155.873, 92.712, 24.669, 178.286]
  MoveL 1128 to (-24.41, -52.55, -272.85) mm, rotated rx 43.39 ry 15.84 rz 65.61 deg; joints [0.024, -1.649, 67.862, 155.926, 92.747, 24.626, 178.286]
  MoveL 1129 to (-26.12, -51.57, -273.06) mm, rotated rx 43.39 ry 15.84 rz 65.61 deg; joints [0.078, -1.6, 67.857, 155.974, 92.779, 24.588, 178.286]
  MoveL 1130 to (-28.18, -50.43, -273.21) mm, rotated rx 43.39 ry 15.84 rz 65.61 deg; joints [0.145, -1.548, 67.858, 156.033, 92.817, 24.541, 178.286]
  MoveL 1131 to (-30.43, -49.19, -273.33) mm, rotated rx 43.39 ry 15.84 rz 65.61 deg; joints [0.218, -1.494, 67.862, 156.097, 92.859, 24.491, 178.286]
  MoveL 1132 to (-32.3, -48.16, -273.33) mm, rotated rx 43.39 ry 15.84 rz 65.61 deg; joints [0.28, -1.455, 67.875, 156.152, 92.895, 24.447, 178.286]
  MoveL 1133 to (-34.07, -47.17, -273.41) mm, rotated rx 43.39 ry 15.84 rz 65.61 deg; joints [0.338, -1.414, 67.88, 156.203, 92.929, 24.407, 178.286]
  MoveL 1134 to (-35.66, -46.26, -273.58) mm, rotated rx 43.39 ry 15.84 rz 65.61 deg; joints [0.389, -1.369, 67.877, 156.248, 92.958, 24.372, 178.286]
  MoveL 1135 to (-37.28, -45.32, -273.79) mm, rotated rx 43.39 ry 15.84 rz 65.61 deg; joints [0.44, -1.322, 67.872, 156.293, 92.989, 24.336, 178.286]
  MoveL 1136 to (-39.34, -44.17, -273.93) mm, rotated rx 43.39 ry 15.84 rz 65.61 deg; joints [0.507, -1.269, 67.872, 156.352, 93.026, 24.29, 178.286]
  MoveL 1137 to (-41.59, -42.91, -274.03) mm, rotated rx 43.39 ry 15.84 rz 65.61 deg; joints [0.581, -1.215, 67.877, 156.417, 93.068, 24.24, 178.286]
  MoveL 1138 to (-45.32, -40.85, -274.03) mm, rotated rx 43.39 ry 15.84 rz 65.61 deg; joints [0.706, -1.137, 67.897, 156.527, 93.139, 24.155, 178.286]
  MoveL 1139 to (-45.4, -40.54, -274.73) mm, rotated rx 43.39 ry 15.84 rz 65.61 deg; joints [0.7, -1.09, 67.858, 156.522, 93.146, 24.155, 178.286]
  MoveL 1140 to (-45.08, -40.57, -275.07) mm, rotated rx 43.39 ry 15.84 rz 65.61 deg; joints [0.685, -1.075, 67.837, 156.509, 93.144, 24.162, 178.286]
  MoveL 1141 to (-45.07, -40.55, -275.29) mm, rotated rx 43.39 ry 15.84 rz 65.61 deg; joints [0.682, -1.06, 67.818, 156.506, 93.141, 24.165, 178.286]
  MoveL 1142 to (-45.33, -40.51, -275.4) mm, rotated rx 43.39 ry 15.84 rz 65.61 deg; joints [0.689, -1.045, 67.8, 156.513, 93.137, 24.163, 178.286]
  MoveL 1143 to (-45.79, -40.49, -275.43) mm, rotated rx 43.39 ry 15.84 rz 65.61 deg; joints [0.703, -1.029, 67.778, 156.525, 93.129, 24.161, 178.286]
  MoveL 1144 to (-46.26, -40.49, -275.46) mm, rotated rx 43.39 ry 15.84 rz 65.61 deg; joints [0.718, -1.012, 67.752, 156.539, 93.119, 24.159, 178.286]
  MoveL 1145 to (-46.7, -40.5, -275.51) mm, rotated rx 43.39 ry 15.84 rz 65.61 deg; joints [0.731, -0.995, 67.727, 156.551, 93.109, 24.158, 178.286]
  MoveL 1146 to (-47.1, -40.5, -275.57) mm, rotated rx 43.39 ry 15.84 rz 65.61 deg; joints [0.743, -0.978, 67.701, 156.562, 93.099, 24.157, 178.286]
  MoveL 1147 to (-47.51, -40.51, -275.63) mm, rotated rx 43.39 ry 15.84 rz 65.61 deg; joints [0.755, -0.961, 67.676, 156.573, 93.09, 24.156, 178.286]
  MoveL 1148 to (-47.95, -40.53, -275.67) mm, rotated rx 43.39 ry 15.84 rz 65.61 deg; joints [0.769, -0.944, 67.649, 156.585, 93.079, 24.154, 178.286]
  MoveL 1149 to (-48.47, -40.56, -275.7) mm, rotated rx 43.39 ry 15.84 rz 65.61 deg; joints [0.785, -0.926, 67.619, 156.6, 93.066, 24.153, 178.286]
  MoveL 1150 to (-49, -40.58, -275.76) mm, rotated rx 43.39 ry 15.84 rz 65.61 deg; joints [0.801, -0.904, 67.587, 156.615, 93.053, 24.152, 178.286]
  MoveL 1151 to (-49.52, -40.6, -275.79) mm, rotated rx 43.39 ry 15.84 rz 65.61 deg; joints [0.817, -0.885, 67.557, 156.629, 93.04, 24.15, 178.286]
  MoveL 1152 to (-50.04, -40.65, -275.8) mm, rotated rx 43.39 ry 15.84 rz 65.61 deg; joints [0.833, -0.868, 67.528, 156.644, 93.027, 24.149, 178.286]
  MoveL 1153 to (-50.56, -40.69, -275.8) mm, rotated rx 43.39 ry 15.84 rz 65.61 deg; joints [0.85, -0.851, 67.499, 156.659, 93.013, 24.148, 178.286]
  MoveL 1154 to (-51.25, -40.77, -275.76) mm, rotated rx 43.39 ry 15.84 rz 65.61 deg; joints [0.872, -0.831, 67.462, 156.68, 92.995, 24.146, 178.286]
  MoveL 1155 to (-51.91, -40.84, -275.73) mm, rotated rx 43.39 ry 15.84 rz 65.61 deg; joints [0.893, -0.811, 67.427, 156.699, 92.977, 24.145, 178.286]
  MoveL 1156 to (-52.51, -40.89, -275.73) mm, rotated rx 43.39 ry 15.84 rz 65.61 deg; joints [0.912, -0.792, 67.394, 156.716, 92.961, 24.143, 178.286]
  MoveL 1157 to (-52.98, -40.91, -275.76) mm, rotated rx 43.39 ry 15.84 rz 65.61 deg; joints [0.926, -0.774, 67.366, 156.729, 92.95, 24.142, 178.286]
  MoveL 1158 to (-53.39, -40.92, -275.82) mm, rotated rx 43.39 ry 15.84 rz 65.61 deg; joints [0.939, -0.757, 67.34, 156.741, 92.94, 24.141, 178.286]
  MoveL 1159 to (-53.8, -40.92, -275.88) mm, rotated rx 43.39 ry 15.84 rz 65.61 deg; joints [0.951, -0.74, 67.315, 156.752, 92.93, 24.14, 178.286]
  MoveL 1160 to (-54.24, -40.94, -275.91) mm, rotated rx 43.39 ry 15.84 rz 65.61 deg; joints [0.965, -0.724, 67.289, 156.764, 92.919, 24.139, 178.286]
  MoveL 1161 to (-55.8, -41.08, -275.91) mm, rotated rx 43.39 ry 15.84 rz 65.61 deg; joints [1.014, -0.672, 67.201, 156.809, 92.878, 24.135, 178.286]
  MoveL 1162 to (-58.69, -41.09, -276.29) mm, rotated rx 43.39 ry 15.84 rz 65.61 deg; joints [1.101, -0.554, 67.024, 156.888, 92.81, 24.126, 178.286]
  MoveL 1163 to (-59.93, -40.91, -276.76) mm, rotated rx 43.39 ry 15.84 rz 65.61 deg; joints [1.134, -0.485, 66.936, 156.919, 92.788, 24.121, 178.286]
  MoveL 1164 to (-61.04, -40.61, -277.42) mm, rotated rx 43.39 ry 15.84 rz 65.61 deg; joints [1.162, -0.408, 66.849, 156.944, 92.774, 24.115, 178.286]
  MoveL 1165 to (-62, -40.18, -278.27) mm, rotated rx 43.39 ry 15.84 rz 65.61 deg; joints [1.183, -0.325, 66.763, 156.963, 92.768, 24.109, 178.286]
  MoveL 1166 to (-62.83, -39.62, -279.3) mm, rotated rx 43.39 ry 15.84 rz 65.61 deg; joints [1.197, -0.234, 66.677, 156.975, 92.77, 24.102, 178.286]
  MoveL 1167 to (-64.08, -38.12, -281.94) mm, rotated rx 43.39 ry 15.84 rz 65.61 deg; joints [1.207, -0.032, 66.506, 156.983, 92.797, 24.086, 178.286]
  MoveL 1168 to (-64.54, -36.6, -284.58) mm, rotated rx 43.39 ry 15.84 rz 65.61 deg; joints [1.191, 0.144, 66.375, 156.969, 92.842, 24.073, 178.286]
  MoveL 1169 to (-64.38, -36.01, -285.61) mm, rotated rx 43.39 ry 15.84 rz 65.61 deg; joints [1.174, 0.203, 66.34, 156.953, 92.866, 24.07, 178.286]
  MoveL 1170 to (-63.96, -35.53, -286.46) mm, rotated rx 43.39 ry 15.84 rz 65.61 deg; joints [1.151, 0.242, 66.325, 156.932, 92.892, 24.07, 178.286]
  MoveL 1171 to (-63.28, -35.16, -287.12) mm, rotated rx 43.39 ry 15.84 rz 65.61 deg; joints [1.122, 0.262, 66.33, 156.905, 92.919, 24.071, 178.286]
  MoveL 1172 to (-62.34, -34.91, -287.59) mm, rotated rx 43.39 ry 15.84 rz 65.61 deg; joints [1.087, 0.261, 66.355, 156.873, 92.947, 24.074, 178.286]
  MoveL 1173 to (-61.14, -34.76, -287.87) mm, rotated rx 43.39 ry 15.84 rz 65.61 deg; joints [1.045, 0.241, 66.4, 156.835, 92.976, 24.079, 178.286]
  MoveL 1174 to (-59.68, -34.73, -287.97) mm, rotated rx 43.39 ry 15.84 rz 65.61 deg; joints [0.998, 0.201, 66.465, 156.792, 93.007, 24.087, 178.286]
  MoveL 1175 to (-59.16, -34.74, -287.97) mm, rotated rx 43.39 ry 15.84 rz 65.61 deg; joints [0.981, 0.185, 66.49, 156.777, 93.017, 24.089, 178.286]
  MoveL 1176 to (-58.69, -34.76, -287.95) mm, rotated rx 43.39 ry 15.84 rz 65.61 deg; joints [0.966, 0.169, 66.513, 156.763, 93.026, 24.092, 178.286]
  MoveL 1177 to (-58.29, -34.79, -287.9) mm, rotated rx 43.39 ry 15.84 rz 65.61 deg; joints [0.954, 0.153, 66.534, 156.752, 93.033, 24.094, 178.286]
  MoveL 1178 to (-57.9, -34.83, -287.84) mm, rotated rx 43.39 ry 15.84 rz 65.61 deg; joints [0.942, 0.138, 66.555, 156.742, 93.04, 24.096, 178.286]
  MoveL 1179 to (-57.47, -34.86, -287.8) mm, rotated rx 43.39 ry 15.84 rz 65.61 deg; joints [0.929, 0.122, 66.577, 156.73, 93.048, 24.099, 178.286]
  MoveL 1180 to (-56.98, -34.88, -287.78) mm, rotated rx 43.39 ry 15.84 rz 65.61 deg; joints [0.914, 0.105, 66.601, 156.716, 93.057, 24.101, 178.286]
  MoveL 1181 to (-56.46, -34.89, -287.78) mm, rotated rx 43.39 ry 15.84 rz 65.61 deg; joints [0.897, 0.088, 66.626, 156.7, 93.067, 24.104, 178.286]
  MoveL 1182 to (-55.99, -34.91, -287.75) mm, rotated rx 43.39 ry 15.84 rz 65.61 deg; joints [0.883, 0.072, 66.649, 156.687, 93.076, 24.107, 178.286]
  MoveL 1183 to (-55.59, -34.93, -287.7) mm, rotated rx 43.39 ry 15.84 rz 65.61 deg; joints [0.87, 0.056, 66.671, 156.676, 93.084, 24.109, 178.286]
  MoveL 1184 to (-55.2, -34.96, -287.64) mm, rotated rx 43.39 ry 15.84 rz 65.61 deg; joints [0.859, 0.04, 66.694, 156.665, 93.091, 24.11, 178.286]
  MoveL 1185 to (-54.77, -34.98, -287.6) mm, rotated rx 43.39 ry 15.84 rz 65.61 deg; joints [0.845, 0.024, 66.717, 156.653, 93.099, 24.113, 178.286]
  MoveL 1186 to (-54.28, -35, -287.57) mm, rotated rx 43.39 ry 15.84 rz 65.61 deg; joints [0.83, 0.007, 66.741, 156.639, 93.109, 24.115, 178.286]
  MoveL 1187 to (-53.75, -35, -287.57) mm, rotated rx 43.39 ry 15.84 rz 65.61 deg; joints [0.813, -0.009, 66.766, 156.624, 93.119, 24.118, 178.286]
  MoveL 1188 to (-52.77, -35.09, -287.55) mm, rotated rx 43.39 ry 15.84 rz 65.61 deg; joints [0.782, -0.04, 66.807, 156.596, 93.133, 24.125, 178.286]
  MoveC 1189 to (-51.4, -35.26, -287.55) mm, rotated rx 43.39 ry 15.84 rz 65.61 deg; joints [0.738, -0.08, 66.857, 156.556, 93.15, 24.137, 178.286] to (-50.02, -35.25, -287.55) mm, rotated rx 43.39 ry 15.84 rz 65.61 deg; joints [0.694, -0.123, 66.924, 156.516, 93.178, 24.144, 178.286]
  MoveL 1190 to (-50.02, -35.25, -287.54) mm, rotated rx 43.39 ry 15.84 rz 65.61 deg; joints [0.694, -0.124, 66.925, 156.516, 93.178, 24.143, 178.286]
  MoveL 1191 to (-49.36, -35.3, -287.52) mm, rotated rx 43.39 ry 15.84 rz 65.61 deg; joints [0.673, -0.145, 66.953, 156.497, 93.188, 24.148, 178.286]
  MoveL 1192 to (-48.8, -35.41, -287.5) mm, rotated rx 43.39 ry 15.84 rz 65.61 deg; joints [0.655, -0.162, 66.972, 156.481, 93.193, 24.154, 178.286]
  MoveL 1193 to (-48.52, -35.53, -287.4) mm, rotated rx 43.39 ry 15.84 rz 65.61 deg; joints [0.647, -0.176, 66.984, 156.474, 93.192, 24.158, 178.286]
  MoveL 1194 to (-48.57, -35.56, -287.2) mm, rotated rx 43.39 ry 15.84 rz 65.61 deg; joints [0.652, -0.188, 66.997, 156.478, 93.193, 24.155, 178.286]
  MoveL 1195 to (-48.99, -35.47, -286.89) mm, rotated rx 43.39 ry 15.84 rz 65.61 deg; joints [0.669, -0.198, 67.015, 156.493, 93.196, 24.146, 178.286]
  MoveL 1196 to (-49.26, -35.75, -286.27) mm, rotated rx 43.39 ry 15.84 rz 65.61 deg; joints [0.685, -0.23, 67.035, 156.508, 93.184, 24.145, 178.286]
  MoveL 1197 to (-47.53, -36.82, -286.26) mm, rotated rx 43.39 ry 15.84 rz 65.61 deg; joints [0.627, -0.265, 67.017, 156.457, 93.144, 24.187, 178.286]
  MoveL 1198 to (-45.76, -38.02, -286.21) mm, rotated rx 43.39 ry 15.84 rz 65.61 deg; joints [0.568, -0.303, 66.993, 156.405, 93.097, 24.233, 178.286]
  MoveL 1199 to (-43.9, -39.33, -286.09) mm, rotated rx 43.39 ry 15.84 rz 65.61 deg; joints [0.507, -0.346, 66.968, 156.351, 93.044, 24.283, 178.286]
  MoveL 1200 to (-42.07, -40.61, -285.98) mm, rotated rx 43.39 ry 15.84 rz 65.61 deg; joints [0.446, -0.386, 66.942, 156.299, 92.993, 24.332, 178.286]
  MoveL 1201 to (-40.31, -41.86, -285.81) mm, rotated rx 43.39 ry 15.84 rz 65.61 deg; joints [0.389, -0.43, 66.923, 156.249, 92.944, 24.378, 178.286]
  MoveL 1202 to (-38.73, -42.98, -285.67) mm, rotated rx 43.39 ry 15.84 rz 65.61 deg; joints [0.338, -0.469, 66.904, 156.204, 92.9, 24.42, 178.286]
  MoveL 1203 to (-37.03, -44.17, -285.61) mm, rotated rx 43.39 ry 15.84 rz 65.61 deg; joints [0.281, -0.504, 66.875, 156.154, 92.851, 24.466, 178.286]
  MoveL 1204 to (-35.26, -45.4, -285.54) mm, rotated rx 43.39 ry 15.84 rz 65.61 deg; joints [0.223, -0.541, 66.847, 156.103, 92.801, 24.514, 178.286]
  MoveL 1205 to (-33.34, -46.75, -285.39) mm, rotated rx 43.39 ry 15.84 rz 65.61 deg; joints [0.16, -0.586, 66.822, 156.048, 92.747, 24.566, 178.286]
  MoveL 1206 to (-31.8, -47.83, -285.27) mm, rotated rx 43.39 ry 15.84 rz 65.61 deg; joints [0.11, -0.621, 66.801, 156.004, 92.703, 24.607, 178.286]
  MoveL 1207 to (-29.84, -49.2, -285.06) mm, rotated rx 43.39 ry 15.84 rz 65.61 deg; joints [0.047, -0.671, 66.781, 155.949, 92.65, 24.659, 178.286]
  MoveL 1208 to (-28.29, -50.27, -284.95) mm, rotated rx 43.39 ry 15.84 rz 65.61 deg; joints [-0.003, -0.707, 66.761, 155.905, 92.607, 24.701, 178.286]
  MoveL 1209 to (-26.54, -51.48, -284.78) mm, rotated rx 43.39 ry 15.84 rz 65.61 deg; joints [-0.06, -0.75, 66.74, 155.855, 92.559, 24.747, 178.286]
  MoveL 1210 to (-24.58, -52.84, -284.73) mm, rotated rx 43.39 ry 15.84 rz 65.61 deg; joints [-0.125, -0.787, 66.704, 155.798, 92.502, 24.802, 178.286]
  MoveL 1211 to (-23.03, -53.91, -284.62) mm, rotated rx 43.39 ry 15.84 rz 65.61 deg; joints [-0.175, -0.822, 66.683, 155.754, 92.459, 24.844, 178.286]
  MoveL 1212 to (-21.27, -55.11, -284.46) mm, rotated rx 43.39 ry 15.84 rz 65.61 deg; joints [-0.232, -0.865, 66.662, 155.705, 92.412, 24.891, 178.286]
  MoveL 1213 to (-19.31, -56.47, -284.41) mm, rotated rx 43.39 ry 15.84 rz 65.61 deg; joints [-0.296, -0.902, 66.625, 155.648, 92.355, 24.946, 178.286]
  MoveL 1214 to (-17.76, -57.53, -284.3) mm, rotated rx 43.39 ry 15.84 rz 65.61 deg; joints [-0.347, -0.937, 66.603, 155.604, 92.312, 24.988, 178.286]
  MoveL 1215 to (-15.92, -58.79, -284.19) mm, rotated rx 43.39 ry 15.84 rz 65.61 deg; joints [-0.406, -0.976, 66.574, 155.552, 92.26, 25.038, 178.286]
  MoveL 1216 to (-14.09, -60.05, -284.13) mm, rotated rx 43.39 ry 15.84 rz 65.61 deg; joints [-0.466, -1.012, 66.541, 155.499, 92.208, 25.09, 178.286]
  MoveL 1217 to (-12.52, -61.08, -283.95) mm, rotated rx 43.39 ry 15.84 rz 65.61 deg; joints [-0.516, -1.052, 66.528, 155.455, 92.168, 25.131, 178.286]
  MoveL 1218 to (-11.06, -62.02, -283.69) mm, rotated rx 43.39 ry 15.84 rz 65.61 deg; joints [-0.561, -1.096, 66.527, 155.416, 92.134, 25.167, 178.286]
  MoveL 1219 to (-9.67, -62.87, -283.34) mm, rotated rx 43.39 ry 15.84 rz 65.61 deg; joints [-0.602, -1.147, 66.54, 155.379, 92.107, 25.198, 178.286]
  MoveL 1220 to (-10.62, -61.7, -282.65) mm, rotated rx 43.39 ry 15.84 rz 65.61 deg; joints [-0.561, -1.191, 66.677, 155.415, 92.184, 25.143, 178.286]
  MoveL 1221 to (-10.46, -61.86, -282.65) mm, rotated rx 43.39 ry 15.84 rz 65.61 deg; joints [-0.566, -1.193, 66.669, 155.41, 92.176, 25.15, 178.286]
  MoveL 1222 to (-10.28, -62.1, -282.63) mm, rotated rx 43.39 ry 15.84 rz 65.61 deg; joints [-0.572, -1.194, 66.655, 155.405, 92.163, 25.158, 178.286]
  MoveL 1223 to (-10.06, -62.5, -282.6) mm, rotated rx 43.39 ry 15.84 rz 65.61 deg; joints [-0.58, -1.195, 66.629, 155.399, 92.139, 25.173, 178.286]
  MoveL 1224 to (-9.83, -62.98, -282.56) mm, rotated rx 43.39 ry 15.84 rz 65.61 deg; joints [-0.588, -1.195, 66.595, 155.392, 92.111, 25.19, 178.286]
  MoveL 1225 to (-9.58, -63.55, -282.52) mm, rotated rx 43.39 ry 15.84 rz 65.61 deg; joints [-0.596, -1.195, 66.556, 155.385, 92.076, 25.209, 178.286]
  MoveL 1226 to (-8.62, -65.99, -282.52) mm, rotated rx 43.39 ry 15.84 rz 65.61 deg; joints [-0.632, -1.175, 66.36, 155.356, 91.923, 25.296, 178.286]
  MoveL 1227 to (-8.39, -66.55, -282.49) mm, rotated rx 43.39 ry 15.84 rz 65.61 deg; joints [-0.64, -1.173, 66.318, 155.349, 91.888, 25.316, 178.286]
  MoveL 1228 to (-8.11, -67.17, -282.43) mm, rotated rx 43.39 ry 15.84 rz 65.61 deg; joints [-0.649, -1.173, 66.274, 155.341, 91.85, 25.337, 178.286]
  MoveL 1229 to (-7.86, -67.75, -282.4) mm, rotated rx 43.39 ry 15.84 rz 65.61 deg; joints [-0.658, -1.171, 66.232, 155.334, 91.815, 25.358, 178.286]
  MoveL 1230 to (-7.67, -68.24, -282.4) mm, rotated rx 43.39 ry 15.84 rz 65.61 deg; joints [-0.665, -1.166, 66.192, 155.329, 91.784, 25.375, 178.286]
  MoveL 1231 to (-7.49, -68.7, -282.39) mm, rotated rx 43.39 ry 15.84 rz 65.61 deg; joints [-0.671, -1.163, 66.156, 155.323, 91.755, 25.391, 178.286]
  MoveL 1232 to (-7.3, -69.18, -282.39) mm, rotated rx 43.39 ry 15.84 rz 65.61 deg; joints [-0.678, -1.159, 66.116, 155.317, 91.724, 25.409, 178.286]
  MoveL 1233 to (-7.11, -69.66, -282.39) mm, rotated rx 43.39 ry 15.84 rz 65.61 deg; joints [-0.685, -1.155, 66.078, 155.312, 91.694, 25.426, 178.286]
  MoveL 1234 to (-6.93, -70.11, -282.36) mm, rotated rx 43.39 ry 15.84 rz 65.61 deg; joints [-0.692, -1.153, 66.044, 155.306, 91.666, 25.442, 178.286]
  MoveL 1235 to (-6.74, -70.53, -282.31) mm, rotated rx 43.39 ry 15.84 rz 65.61 deg; joints [-0.698, -1.154, 66.015, 155.301, 91.641, 25.456, 178.286]
  MoveL 1236 to (-6.55, -70.99, -282.3) mm, rotated rx 43.39 ry 15.84 rz 65.61 deg; joints [-0.705, -1.151, 65.98, 155.295, 91.612, 25.473, 178.286]
  MoveL 1237 to (-6.36, -71.49, -282.29) mm, rotated rx 43.39 ry 15.84 rz 65.61 deg; joints [-0.712, -1.147, 65.94, 155.29, 91.581, 25.49, 178.286]
  MoveL 1238 to (-5.97, -72.46, -282.29) mm, rotated rx 43.39 ry 15.84 rz 65.61 deg; joints [-0.726, -1.138, 65.86, 155.278, 91.519, 25.525, 178.286]
  Set speed (1000.0 mm/s)
  MoveL 1239 to (-4.09, -94, -282.29) mm, rotated rx 43.39 ry 15.84 rz 65.61 deg; joints [-0.827, -0.712, 63.753, 155.197, 90.011, 26.27, 178.286]
  Print: /'Flow1'
  Set speed (1000.0 mm/s)
  MoveL 1240 to (115.79, 27.59, -71.8) mm, rotated rx -11.83 ry -17.7 rz 126.62 deg; joints [4.247, -43.756, 123.216, 233.375, 67.797, -46.528, 143.741]
  Set speed (1000.0 mm/s)
  MoveL 1241 to (75.12, 46.55, -71.8) mm, rotated rx -11.83 ry -17.7 rz 126.62 deg; joints [6.14, -43.497, 124.253, 234.899, 68.82, -45.603, 143.741]
  Set speed (100.0 mm/s)
  MoveL 1242 to (9.17, 77.31, -71.8) mm, rotated rx -11.83 ry -17.7 rz 126.62 deg; joints [9.303, -42.945, 125.661, 237.516, 70.288, -44.134, 143.741]
  MoveL 1243 to (8.93, 77.77, -71.8) mm, rotated rx -11.83 ry -17.7 rz 126.62 deg; joints [9.318, -42.956, 125.693, 237.525, 70.3, -44.117, 143.741]
  MoveL 1244 to (8.6, 78.32, -71.7) mm, rotated rx -11.83 ry -17.7 rz 126.62 deg; joints [9.34, -42.974, 125.729, 237.542, 70.313, -44.102, 143.741]
  MoveL 1245 to (8.3, 78.83, -71.65) mm, rotated rx -11.83 ry -17.7 rz 126.62 deg; joints [9.36, -42.988, 125.764, 237.556, 70.325, -44.085, 143.741]
  MoveL 1246 to (8.03, 79.33, -71.62) mm, rotated rx -11.83 ry -17.7 rz 126.62 deg; joints [9.377, -43.001, 125.798, 237.567, 70.339, -44.068, 143.741]
  MoveL 1247 to (6.37, 82.6, -71.62) mm, rotated rx -11.83 ry -17.7 rz 126.62 deg; joints [9.486, -43.081, 126.024, 237.634, 70.428, -43.945, 143.741]
  MoveL 1248 to (5.77, 83.92, -71.71) mm, rotated rx -11.83 ry -17.7 rz 126.62 deg; joints [9.526, -43.11, 126.117, 237.655, 70.467, -43.89, 143.741]
  MoveL 1249 to (5.41, 85.05, -71.98) mm, rotated rx -11.83 ry -17.7 rz 126.62 deg; joints [9.551, -43.128, 126.2, 237.661, 70.504, -43.833, 143.741]
  MoveL 1250 to (5.27, 85.99, -72.42) mm, rotated rx -11.83 ry -17.7 rz 126.62 deg; joints [9.562, -43.134, 126.273, 237.652, 70.541, -43.773, 143.741]
  MoveL 1251 to (5.29, 86.39, -72.71) mm, rotated rx -11.83 ry -17.7 rz 126.62 deg; joints [9.562, -43.133, 126.306, 237.641, 70.56, -43.743, 143.741]
  MoveL 1252 to (5.37, 86.73, -73.04) mm, rotated rx -11.83 ry -17.7 rz 126.62 deg; joints [9.558, -43.129, 126.337, 237.627, 70.578, -43.711, 143.741]
  MoveL 1253 to (5.7, 87.29, -73.84) mm, rotated rx -11.83 ry -17.7 rz 126.62 deg; joints [9.539, -43.112, 126.391, 237.587, 70.614, -43.647, 143.741]
  MoveL 1254 to (6.26, 87.65, -74.82) mm, rotated rx -11.83 ry -17.7 rz 126.62 deg; joints [9.505, -43.084, 126.436, 237.531, 70.649, -43.58, 143.741]
  MoveL 1255 to (8.08, 87.8, -77.3) mm, rotated rx -11.83 ry -17.7 rz 126.62 deg; joints [9.393, -42.995, 126.496, 237.373, 70.719, -43.439, 143.741]
  MoveL 1256 to (10.22, 87.23, -79.79) mm, rotated rx -11.83 ry -17.7 rz 126.62 deg; joints [9.258, -42.886, 126.504, 237.202, 70.77, -43.326, 143.741]
  MoveL 1257 to (12.07, 85.96, -81.56) mm, rotated rx -11.83 ry -17.7 rz 126.62 deg; joints [9.139, -42.784, 126.448, 237.068, 70.783, -43.277, 143.741]
  MoveL 1258 to (12.88, 85.08, -82.18) mm, rotated rx -11.83 ry -17.7 rz 126.62 deg; joints [9.085, -42.737, 126.397, 237.014, 70.776, -43.277, 143.741]
  MoveL 1259 to (13.61, 84.02, -82.63) mm, rotated rx -11.83 ry -17.7 rz 126.62 deg; joints [9.035, -42.691, 126.33, 236.969, 70.76, -43.293, 143.741]
  MoveL 1260 to (14.86, 81.38, -82.98) mm, rotated rx -11.83 ry -17.7 rz 126.62 deg; joints [8.947, -42.605, 126.148, 236.908, 70.7, -43.372, 143.741]
  MoveL 1261 to (15.96, 78.43, -82.99) mm, rotated rx -11.83 ry -17.7 rz 126.62 deg; joints [8.867, -42.522, 125.936, 236.865, 70.621, -43.482, 143.741]
  MoveL 1262 to (16.14, 77.98, -83.01) mm, rotated rx -11.83 ry -17.7 rz 126.62 deg; joints [8.854, -42.509, 125.904, 236.857, 70.61, -43.498, 143.741]
  MoveL 1263 to (16.32, 77.55, -83.05) mm, rotated rx -11.83 ry -17.7 rz 126.62 deg; joints [8.841, -42.496, 125.874, 236.848, 70.599, -43.512, 143.741]
  MoveL 1264 to (16.5, 77.18, -83.11) mm, rotated rx -11.83 ry -17.7 rz 126.62 deg; joints [8.828, -42.483, 125.848, 236.839, 70.591, -43.522, 143.741]
  MoveL 1265 to (16.69, 76.77, -83.16) mm, rotated rx -11.83 ry -17.7 rz 126.62 deg; joints [8.815, -42.47, 125.82, 236.83, 70.582, -43.535, 143.741]
  MoveL 1266 to (16.89, 76.27, -83.18) mm, rotated rx -11.83 ry -17.7 rz 126.62 deg; joints [8.8, -42.455, 125.784, 236.822, 70.569, -43.552, 143.741]
  MoveL 1267 to (17.14, 75.67, -83.22) mm, rotated rx -11.83 ry -17.7 rz 126.62 deg; joints [8.782, -42.436, 125.741, 236.811, 70.554, -43.573, 143.741]
  MoveL 1268 to (17.36, 75.15, -83.28) mm, rotated rx -11.83 ry -17.7 rz 126.62 deg; joints [8.766, -42.42, 125.706, 236.8, 70.542, -43.589, 143.741]
  MoveL 1269 to (17.56, 74.75, -83.35) mm, rotated rx -11.83 ry -17.7 rz 126.62 deg; joints [8.752, -42.405, 125.678, 236.79, 70.533, -43.6, 143.741]
  MoveL 1270 to (17.74, 74.35, -83.4) mm, rotated rx -11.83 ry -17.7 rz 126.62 deg; joints [8.74, -42.392, 125.65, 236.782, 70.524, -43.612, 143.741]
  MoveL 1271 to (17.91, 73.91, -83.43) mm, rotated rx -11.83 ry -17.7 rz 126.62 deg; joints [8.727, -42.379, 125.618, 236.774, 70.512, -43.627, 143.741]
  MoveL 1272 to (18.1, 73.42, -83.43) mm, rotated rx -11.83 ry -17.7 rz 126.62 deg; joints [8.714, -42.365, 125.583, 236.767, 70.499, -43.646, 143.741]
  MoveL 1273 to (18.29, 72.91, -83.43) mm, rotated rx -11.83 ry -17.7 rz 126.62 deg; joints [8.7, -42.351, 125.546, 236.76, 70.486, -43.664, 143.741]
  MoveL 1274 to (18.5, 72.38, -83.44) mm, rotated rx -11.83 ry -17.7 rz 126.62 deg; joints [8.685, -42.336, 125.508, 236.751, 70.472, -43.684, 143.741]
  MoveL 1275 to (18.76, 71.77, -83.47) mm, rotated rx -11.83 ry -17.7 rz 126.62 deg; joints [8.667, -42.318, 125.465, 236.74, 70.456, -43.705, 143.741]
  MoveL 1276 to (19.02, 71.24, -83.54) mm, rotated rx -11.83 ry -17.7 rz 126.62 deg; joints [8.649, -42.301, 125.429, 236.728, 70.443, -43.721, 143.741]
  MoveL 1277 to (19.25, 70.85, -83.64) mm, rotated rx -11.83 ry -17.7 rz 126.62 deg; joints [8.634, -42.286, 125.402, 236.716, 70.435, -43.731, 143.741]
  MoveL 1278 to (19.24, 70.84, -83.88) mm, rotated rx -11.83 ry -17.7 rz 126.62 deg; joints [8.631, -42.272, 125.403, 236.708, 70.443, -43.717, 143.741]
  MoveL 1279 to (18.99, 71.15, -84.23) mm, rotated rx -11.83 ry -17.7 rz 126.62 deg; joints [8.64, -42.256, 125.425, 236.707, 70.465, -43.684, 143.741]
  MoveL 1280 to (19.19, 71.98, -85.2) mm, rotated rx -11.83 ry -17.7 rz 126.62 deg; joints [8.627, -42.237, 125.498, 236.666, 70.514, -43.601, 143.741]
  MoveL 1281 to (20.92, 70.73, -85.2) mm, rotated rx -11.83 ry -17.7 rz 126.62 deg; joints [8.538, -42.237, 125.43, 236.596, 70.468, -43.655, 143.741]
  MoveL 1282 to (22.8, 69.41, -85.33) mm, rotated rx -11.83 ry -17.7 rz 126.62 deg; joints [8.44, -42.23, 125.359, 236.516, 70.423, -43.706, 143.741]
  MoveL 1283 to (24.57, 68.14, -85.38) mm, rotated rx -11.83 ry -17.7 rz 126.62 deg; joints [8.349, -42.226, 125.289, 236.443, 70.377, -43.758, 143.741]
  MoveL 1284 to (26.31, 66.92, -85.52) mm, rotated rx -11.83 ry -17.7 rz 126.62 deg; joints [8.259, -42.219, 125.222, 236.369, 70.336, -43.804, 143.741]
  MoveL 1285 to (28.05, 65.68, -85.67) mm, rotated rx -11.83 ry -17.7 rz 126.62 deg; joints [8.168, -42.21, 125.155, 236.294, 70.294, -43.849, 143.741]
  MoveL 1286 to (29.78, 64.45, -85.79) mm, rotated rx -11.83 ry -17.7 rz 126.62 deg; joints [8.079, -42.202, 125.087, 236.221, 70.251, -43.896, 143.741]
  MoveL 1287 to (31.53, 63.21, -86) mm, rotated rx -11.83 ry -17.7 rz 126.62 deg; joints [7.987, -42.19, 125.018, 236.145, 70.211, -43.938, 143.741]
  MoveL 1288 to (33.26, 61.97, -86.12) mm, rotated rx -11.83 ry -17.7 rz 126.62 deg; joints [7.898, -42.182, 124.95, 236.072, 70.167, -43.986, 143.741]
  MoveL 1289 to (35, 60.71, -86.17) mm, rotated rx -11.83 ry -17.7 rz 126.62 deg; joints [7.809, -42.177, 124.879, 236.002, 70.121, -44.037, 143.741]
  MoveL 1290 to (36.75, 59.45, -86.32) mm, rotated rx -11.83 ry -17.7 rz 126.62 deg; joints [7.719, -42.167, 124.808, 235.928, 70.077, -44.084, 143.741]
  MoveL 1291 to (38.56, 58.15, -86.5) mm, rotated rx -11.83 ry -17.7 rz 126.62 deg; joints [7.625, -42.155, 124.735, 235.851, 70.033, -44.131, 143.741]
  MoveL 1292 to (40.36, 56.85, -86.68) mm, rotated rx -11.83 ry -17.7 rz 126.62 deg; joints [7.532, -42.143, 124.66, 235.774, 69.988, -44.177, 143.741]
  MoveL 1293 to (41.87, 55.74, -86.92) mm, rotated rx -11.83 ry -17.7 rz 126.62 deg; joints [7.453, -42.126, 124.598, 235.707, 69.954, -44.212, 143.741]
  MoveL 1294 to (44.03, 54.17, -87.03) mm, rotated rx -11.83 ry -17.7 rz 126.62 deg; joints [7.343, -42.117, 124.508, 235.62, 69.896, -44.274, 143.741]
  Set speed (1000.0 mm/s)
  MoveL 1295 to (85.09, 35.03, -87.03) mm, rotated rx -11.83 ry -17.7 rz 126.62 deg; joints [5.404, -42.436, 123.557, 234.03, 68.938, -45.212, 143.741]
  Set speed (1000.0 mm/s)
  MoveL 1296 to (82.67, 29.83, -98.91) mm, rotated rx -11.83 ry -17.7 rz 126.62 deg; joints [5.3, -41.499, 123.17, 233.755, 69.249, -44.726, 143.741]
  Set speed (100.0 mm/s)
  MoveL 1297 to (56.67, 41.95, -98.91) mm, rotated rx -11.83 ry -17.7 rz 126.62 deg; joints [6.521, -41.299, 123.784, 234.754, 69.862, -44.126, 143.741]
  MoveL 1298 to (55.43, 43.14, -98.66) mm, rotated rx -11.83 ry -17.7 rz 126.62 deg; joints [6.588, -41.326, 123.86, 234.808, 69.897, -44.089, 143.741]
  MoveL 1299 to (53.95, 44.52, -98.6) mm, rotated rx -11.83 ry -17.7 rz 126.62 deg; joints [6.665, -41.344, 123.947, 234.866, 69.945, -44.034, 143.741]
  MoveL 1300 to (52.44, 45.92, -98.45) mm, rotated rx -11.83 ry -17.7 rz 126.62 deg; joints [6.745, -41.366, 124.036, 234.927, 69.991, -43.983, 143.741]
  MoveL 1301 to (50.65, 47.6, -98.32) mm, rotated rx -11.83 ry -17.7 rz 126.62 deg; joints [6.839, -41.391, 124.143, 234.999, 70.048, -43.919, 143.741]
  MoveL 1302 to (49.08, 49.05, -98.32) mm, rotated rx -11.83 ry -17.7 rz 126.62 deg; joints [6.92, -41.405, 124.234, 235.059, 70.101, -43.858, 143.741]
  MoveL 1303 to (47.35, 50.65, -98.16) mm, rotated rx -11.83 ry -17.7 rz 126.62 deg; joints [7.012, -41.43, 124.334, 235.13, 70.154, -43.799, 143.741]
  MoveL 1304 to (45.89, 52.01, -97.98) mm, rotated rx -11.83 ry -17.7 rz 126.62 deg; joints [7.091, -41.453, 124.419, 235.192, 70.196, -43.752, 143.741]
  MoveL 1305 to (44.39, 53.4, -97.88) mm, rotated rx -11.83 ry -17.7 rz 126.62 deg; joints [7.17, -41.472, 124.506, 235.252, 70.243, -43.698, 143.741]
  MoveL 1306 to (42.82, 54.84, -97.67) mm, rotated rx -11.83 ry -17.7 rz 126.62 deg; joints [7.255, -41.498, 124.595, 235.32, 70.288, -43.649, 143.741]
  MoveL 1307 to (41.26, 56.27, -97.51) mm, rotated rx -11.83 ry -17.7 rz 126.62 deg; joints [7.338, -41.52, 124.683, 235.385, 70.333, -43.597, 143.741]
  MoveL 1308 to (39.7, 57.7, -97.4) mm, rotated rx -11.83 ry -17.7 rz 126.62 deg; joints [7.421, -41.539, 124.771, 235.449, 70.381, -43.542, 143.741]
  MoveL 1309 to (38.12, 59.14, -97.23) mm, rotated rx -11.83 ry -17.7 rz 126.62 deg; joints [7.506, -41.561, 124.859, 235.516, 70.426, -43.49, 143.741]
  MoveL 1310 to (36.54, 60.57, -97.09) mm, rotated rx -11.83 ry -17.7 rz 126.62 deg; joints [7.591, -41.581, 124.947, 235.582, 70.472, -43.438, 143.741]
  MoveL 1311 to (34.94, 62.04, -97.02) mm, rotated rx -11.83 ry -17.7 rz 126.62 deg; joints [7.676, -41.597, 125.037, 235.647, 70.522, -43.379, 143.741]
  MoveL 1312 to (33.35, 63.46, -96.81) mm, rotated rx -11.83 ry -17.7 rz 126.62 deg; joints [7.762, -41.62, 125.122, 235.717, 70.566, -43.33, 143.741]
  MoveL 1313 to (31.78, 64.88, -96.69) mm, rotated rx -11.83 ry -17.7 rz 126.62 deg; joints [7.847, -41.639, 125.208, 235.783, 70.611, -43.277, 143.741]
  MoveL 1314 to (30.17, 66.33, -96.57) mm, rotated rx -11.83 ry -17.7 rz 126.62 deg; joints [7.933, -41.657, 125.296, 235.851, 70.658, -43.222, 143.741]
  MoveL 1315 to (28.77, 67.42, -96.36) mm, rotated rx -11.83 ry -17.7 rz 126.62 deg; joints [8.008, -41.673, 125.357, 235.913, 70.691, -43.186, 143.741]
  MoveL 1316 to (27.53, 68.21, -96.01) mm, rotated rx -11.83 ry -17.7 rz 126.62 deg; joints [8.075, -41.689, 125.397, 235.975, 70.71, -43.17, 143.741]
  MoveL 1317 to (26.42, 68.69, -95.48) mm, rotated rx -11.83 ry -17.7 rz 126.62 deg; joints [8.136, -41.708, 125.414, 236.037, 70.714, -43.176, 143.741]
